KUKA KRL program: EPS_2_25999_MH3A_A_20251114084356.src

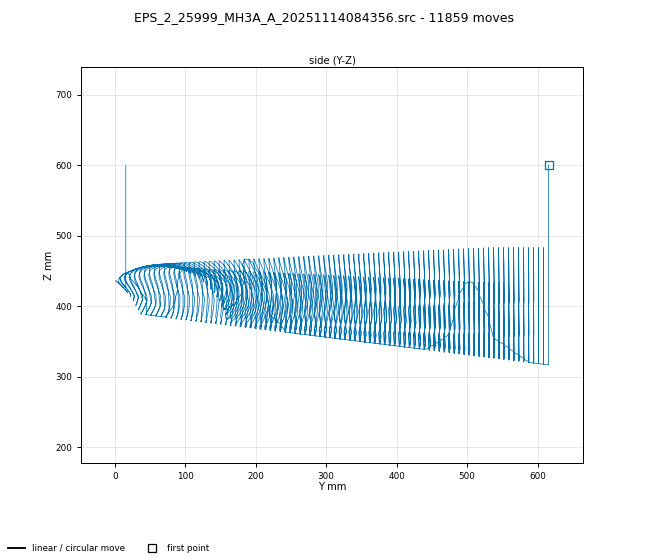
[picture p0: tool path of EPS_2_25999_MH3A_A_20251114084356.src, 11859 of 11861 moves have a stored position in this frame; points joined in program order, loops and branches not executed]
&ACCESS RVP
&REL 4
&COMMENT QRS 19112012
&PARAM EDITMASK = *
DEF PART()
EXT BAS (BAS_COMMAND :IN,REAL :IN )
INT I
BAS (#INITMOV,0 )

;KUKA QRS Post kuka4.cps  Date:22-06-2017 !

File_ID=2914

QRS_PRE_INIT()

;Init var - Until changes are made in qrs_pre_init
Outlet_Square_prg=0
Inlet_1_Square_prg=0
Inlet_2_Square_prg=0
Inlet_3_Square_prg=0
Inlet_4_Square_prg=0
Inlet_5_Square_prg=0

Outlet_1={X 0.000, Y 530.910, Z 408.000, B 0.000, E1 0.000 }
Inlet_1={X 0.000, Y 534.490, Z 358.000, B 0.000, E1 140.000 }
Outlet_1_type=150
Inlet_1_type=150
;QRS#1=Sidecore dimensions
;QRS#2=150-6" PVC SDR 28
;QRS#3=150-6" PVC SDR 28
;QRS#4=
;QRS#5=
;QRS#6=
;QRS#7=
;QRS#8=
;QRS#9=10-06 PSX
;QRS#10=10-06 PSX
;QRS#11=
;QRS#12=
;QRS#13=
;QRS#14=
;QRS#15=
;QRS#16=1220x127x762 2,5'
;QRS#17=EPS Height
;QRS#18=483
;QRS#19=*
;QRS#20= UPDATED VERSION 22-06-2017
;QRS#21=*
Outlet_Square=070
Inlet_1_Square=070
Inlet_2_Square=0
Inlet_3_Square=0
Inlet_4_Square=0
Inlet_5_Square=0
Mill_Square=1
Outlet_Square_Prg=203
Inlet_1_Square_prg=203

QRS_INIT()

$ADVANCE=5

; T1
PTP {E1 173.609,E2 173.609}
PTP {X 0,Y 615.506,A -85,B 0,C 180,E1 173.609,E2 173.609,E3 0,E4 0,E5 0,E6 0}
QRS_SPEED_INIT()
LIN {X 0,Y 615.506,Z 600,A -85,B 0,C 180,E1 173.609,E2 173.609,E3 0,E4 0,E5 0,E6 0} C_VEL
LIN {X 0,Y 615.506,Z 326.684,A -85,B 0,C 180,E1 173.609,E2 173.609} C_VEL
LIN {X 0,Y 615.506,Z 318.507,A -85,B 0,C 180,E1 173.609,E2 173.609} C_VEL
LIN {X 0,Y 615.491,Z 316.507,A -85,B 0,C 180,E1 173.422,E2 173.422} C_VEL
LIN {X 0,Y 615.476,Z 316.513,A -85,B 0,C 180,E1 170.802,E2 170.802} C_VEL
LIN {X 0,Y 615.489,Z 316.515,A -85,B 0,C 180,E1 168.14,E2 168.14} C_VEL
LIN {X 0,Y 615.477,Z 316.512,A -85,B 0,C 180,E1 165.452,E2 165.452} C_VEL
LIN {X 0,Y 615.469,Z 316.512,A -85,B 0,C 180,E1 162.73,E2 162.73} C_VEL
LIN {X 0,Y 615.495,Z 317.045,A -85,B 0,C 180,E1 162.044,E2 162.044} C_VEL
LIN {X 0,Y 615.473,Z 321.165,A -85,B 0,C 180,E1 159.27,E2 159.27} C_VEL
LIN {X 0,Y 615.483,Z 324.407,A -85,B 0,C 180,E1 157.156,E2 157.156} C_VEL
LIN {X 0,Y 615.467,Z 328.675,A -85,B 0,C 180,E1 154.436,E2 154.436} C_VEL
LIN {X 0,Y 615.496,Z 333.308,A -85,B 0,C 180,E1 151.549,E2 151.549} C_VEL
LIN {X 0,Y 615.434,Z 337.615,A -85,B 0,C 180,E1 148.923,E2 148.923} C_VEL
LIN {X 0,Y 615.452,Z 341.695,A -85,B 0,C 180,E1 146.472,E2 146.472} C_VEL
LIN {X 0,Y 615.447,Z 346.56,A -85,B 0,C 180,E1 143.574,E2 143.574} C_VEL
LIN {X 0,Y 615.469,Z 351.05,A -85,B 0,C 180,E1 140.941,E2 140.941} C_VEL
LIN {X 0,Y 615.479,Z 354.222,A -85,B 0,C 180,E1 139.089,E2 139.089} C_VEL
LIN {X 0,Y 615.488,Z 365.834,A -85,B 0,C 180,E1 138.765,E2 138.765} C_VEL
LIN {X 0,Y 615.49,Z 374.096,A -85,B 0,C 180,E1 138.452,E2 138.452} C_VEL
LIN {X 0,Y 615.489,Z 381.984,A -85,B 0,C 180,E1 138.074,E2 138.074} C_VEL
LIN {X 0,Y 615.47,Z 390.539,A -85,B 0,C 180,E1 137.56,E2 137.56} C_VEL
LIN {X 0,Y 615.499,Z 397.606,A -85,B 0,C 180,E1 137.04,E2 137.04} C_VEL
LIN {X 0,Y 615.497,Z 404.982,A -85,B 0,C 180,E1 136.381,E2 136.381} C_VEL
LIN {X 0,Y 615.495,Z 411.606,A -85,B 0,C 180,E1 135.657,E2 135.657} C_VEL
LIN {X 0,Y 615.495,Z 418.335,A -85,B 0,C 180,E1 134.737,E2 134.737} C_VEL
LIN {X 0,Y 615.493,Z 422.558,A -85,B 0,C 180,E1 134,E2 134} C_VEL
LIN {X 0,Y 615.491,Z 426.704,A -85,B 0,C 180,E1 133.049,E2 133.049} C_VEL
LIN {X 0,Y 615.494,Z 429.688,A -85,B 0,C 180,E1 132.082,E2 132.082} C_VEL
LIN {X 0,Y 615.49,Z 431.568,A -85,B 0,C 180,E1 131.097,E2 131.097} C_VEL
LIN {X 0,Y 615.495,Z 432.347,A -85,B 0,C 180,E1 130.092,E2 130.092} C_VEL
LIN {X 0,Y 615.488,Z 431.699,A -85,B 0,C 180,E1 128.905,E2 128.905} C_VEL
LIN {X 0,Y 615.492,Z 430.141,A -85,B 0,C 180,E1 128.014,E2 128.014} C_VEL
LIN {X 0,Y 615.491,Z 426.975,A -85,B 0,C 180,E1 126.939,E2 126.939} C_VEL
LIN {X 0,Y 615.494,Z 422.174,A -85,B 0,C 180,E1 125.837,E2 125.837} C_VEL
LIN {X 0,Y 615.494,Z 417.278,A -85,B 0,C 180,E1 125.015,E2 125.015} C_VEL
LIN {X 0,Y 615.497,Z 411.085,A -85,B 0,C 180,E1 124.192,E2 124.192} C_VEL
LIN {X 0,Y 615.496,Z 405.073,A -85,B 0,C 180,E1 123.538,E2 123.538} C_VEL
LIN {X 0,Y 615.498,Z 398.504,A -85,B 0,C 180,E1 122.943,E2 122.943} C_VEL
LIN {X 0,Y 615.493,Z 392.117,A -85,B 0,C 180,E1 122.458,E2 122.458} C_VEL
LIN {X 0,Y 615.459,Z 385.126,A -85,B 0,C 180,E1 122.01,E2 122.01} C_VEL
LIN {X 0,Y 615.457,Z 375.902,A -85,B 0,C 180,E1 121.538,E2 121.538} C_VEL
LIN {X 0,Y 615.476,Z 367.411,A -85,B 0,C 180,E1 121.199,E2 121.199} C_VEL
LIN {X 0,Y 615.486,Z 359.644,A -85,B 0,C 180,E1 120.962,E2 120.962} C_VEL
LIN {X 0,Y 615.494,Z 354.226,A -85,B 0,C 180,E1 120.825,E2 120.825} C_VEL
LIN {X 0,Y 615.471,Z 349.24,A -85,B 0,C 180,E1 117.917,E2 117.917} C_VEL
LIN {X 0,Y 615.495,Z 345.264,A -85,B 0,C 180,E1 115.573,E2 115.573} C_VEL
LIN {X 0,Y 615.478,Z 340.687,A -85,B 0,C 180,E1 112.846,E2 112.846} C_VEL
LIN {X 0,Y 615.482,Z 336.043,A -85,B 0,C 180,E1 110.034,E2 110.034} C_VEL
LIN {X 0,Y 615.452,Z 332.672,A -85,B 0,C 180,E1 107.959,E2 107.959} C_VEL
LIN {X 0,Y 615.43,Z 329.378,A -85,B 0,C 180,E1 105.907,E2 105.907} C_VEL
LIN {X 0,Y 615.459,Z 325.104,A -85,B 0,C 180,E1 103.203,E2 103.203} C_VEL
LIN {X 0,Y 615.473,Z 320.993,A -85,B 0,C 180,E1 100.528,E2 100.528} C_VEL
LIN {X 0,Y 615.482,Z 317.044,A -85,B 0,C 180,E1 97.876,E2 97.876} C_VEL
LIN {X 0,Y 615.483,Z 316.509,A -85,B 0,C 180,E1 97.216,E2 97.216} C_VEL
LIN {X 0,Y 615.479,Z 316.51,A -85,B 0,C 180,E1 94.585,E2 94.585} C_VEL
LIN {X 0,Y 615.471,Z 316.512,A -85,B 0,C 180,E1 91.964,E2 91.964} C_VEL
LIN {X 0,Y 615.483,Z 316.512,A -85,B 0,C 180,E1 89.347,E2 89.347} C_VEL
LIN {X 0,Y 615.49,Z 316.514,A -85,B 0,C 180,E1 86.728,E2 86.728} C_VEL
LIN {X 0,Y 615.481,Z 316.512,A -85,B 0,C 180,E1 84.102,E2 84.102} C_VEL
LIN {X 0,Y 615.485,Z 316.509,A -85,B 0,C 180,E1 81.464,E2 81.464} C_VEL
LIN {X 0,Y 615.477,Z 316.51,A -85,B 0,C 180,E1 78.808,E2 78.808} C_VEL
LIN {X 0,Y 615.478,Z 316.512,A -85,B 0,C 180,E1 76.066,E2 76.066} C_VEL
LIN {X 0,Y 615.492,Z 316.514,A -85,B 0,C 180,E1 73.415,E2 73.415} C_VEL
LIN {X 0,Y 615.475,Z 316.512,A -85,B 0,C 180,E1 70.663,E2 70.663} C_VEL
LIN {X 0,Y 615.497,Z 316.512,A -85,B 0,C 180,E1 68.57,E2 68.57} C_VEL
LIN {X 0,Y 615.489,Z 316.508,A -85,B 0,C 180,E1 65.729,E2 65.729} C_VEL
LIN {X 0,Y 615.479,Z 316.511,A -85,B 0,C 180,E1 62.824,E2 62.824} C_VEL
LIN {X 0,Y 615.484,Z 316.512,A -85,B 0,C 180,E1 60.204,E2 60.204} C_VEL
LIN {X 0,Y 615.495,Z 316.512,A -85,B 0,C 180,E1 57.544,E2 57.544} C_VEL
LIN {X 0,Y 615.498,Z 316.513,A -85,B 0,C 180,E1 55.187,E2 55.187} C_VEL
LIN {X 0,Y 615.49,Z 316.515,A -85,B 0,C 180,E1 52.759,E2 52.759} C_VEL
LIN {X 0,Y 615.489,Z 316.508,A -85,B 0,C 180,E1 49.909,E2 49.909} C_VEL
LIN {X 0,Y 615.477,Z 316.512,A -85,B 0,C 180,E1 46.952,E2 46.952} C_VEL
LIN {X 0,Y 615.494,Z 316.509,A -85,B 0,C 180,E1 44,E2 44} C_VEL
LIN {X 0,Y 615.468,Z 316.512,A -85,B 0,C 180,E1 41.094,E2 41.094} C_VEL
LIN {X 0,Y 615.467,Z 316.513,A -85,B 0,C 180,E1 38.905,E2 38.905} C_VEL
LIN {X 0,Y 615.474,Z 316.511,A -85,B 0,C 180,E1 36.424,E2 36.424} C_VEL
LIN {X 0,Y 615.492,Z 316.51,A -85,B 0,C 180,E1 33.537,E2 33.537} C_VEL
LIN {X 0,Y 615.491,Z 316.514,A -85,B 0,C 180,E1 30.918,E2 30.918} C_VEL
LIN {X 0,Y 615.496,Z 316.513,A -85,B 0,C 180,E1 28.454,E2 28.454} C_VEL
LIN {X 0,Y 615.466,Z 316.513,A -85,B 0,C 180,E1 25.568,E2 25.568} C_VEL
LIN {X 0,Y 615.468,Z 316.512,A -85,B 0,C 180,E1 22.844,E2 22.844} C_VEL
LIN {X 0,Y 615.493,Z 316.513,A -85,B 0,C 180,E1 20.032,E2 20.032} C_VEL
LIN {X 0,Y 615.476,Z 316.512,A -85,B 0,C 180,E1 17.27,E2 17.27} C_VEL
LIN {X 0,Y 615.485,Z 316.508,A -85,B 0,C 180,E1 14.548,E2 14.548} C_VEL
LIN {X 0,Y 615.484,Z 316.509,A -85,B 0,C 180,E1 11.86,E2 11.86} C_VEL
LIN {X 0,Y 615.483,Z 316.513,A -85,B 0,C 180,E1 9.198,E2 9.198} C_VEL
LIN {X 0,Y 615.494,Z 316.512,A -85,B 0,C 180,E1 6.556,E2 6.556} C_VEL
LIN {X 0,Y 615.477,Z 316.512,A -85,B 0,C 180,E1 3.928,E2 3.928} C_VEL
LIN {X 0,Y 615.468,Z 316.512,A -85,B 0,C 180,E1 1.308,E2 1.308} C_VEL
LIN {X 0,Y 615.49,Z 316.507,A -85,B 0,C 180,E1 -1.309,E2 -1.309} C_VEL
LIN {X 0,Y 615.483,Z 316.51,A -85,B 0,C 180,E1 -3.929,E2 -3.929} C_VEL
LIN {X 0,Y 615.482,Z 316.513,A -85,B 0,C 180,E1 -6.585,E2 -6.585} C_VEL
LIN {X 0,Y 615.496,Z 316.513,A -85,B 0,C 180,E1 -9.199,E2 -9.199} C_VEL
LIN {X 0,Y 615.477,Z 316.512,A -85,B 0,C 180,E1 -11.862,E2 -11.862} C_VEL
LIN {X 0,Y 615.466,Z 316.512,A -85,B 0,C 180,E1 -14.55,E2 -14.55} C_VEL
LIN {X 0,Y 615.496,Z 316.507,A -85,B 0,C 180,E1 -17.271,E2 -17.271} C_VEL
LIN {X 0,Y 615.49,Z 316.513,A -85,B 0,C 180,E1 -20.033,E2 -20.033} C_VEL
LIN {X 0,Y 615.492,Z 316.508,A -85,B 0,C 180,E1 -22.845,E2 -22.845} C_VEL
LIN {X 0,Y 615.472,Z 316.512,A -85,B 0,C 180,E1 -25.717,E2 -25.717} C_VEL
LIN {X 0,Y 615.484,Z 316.513,A -85,B 0,C 180,E1 -28.452,E2 -28.452} C_VEL
LIN {X 0,Y 615.482,Z 316.515,A -85,B 0,C 180,E1 -31.088,E2 -31.088} C_VEL
LIN {X 0,Y 615.491,Z 316.512,A -85,B 0,C 180,E1 -33.537,E2 -33.537} C_VEL
LIN {X 0,Y 615.491,Z 316.514,A -85,B 0,C 180,E1 -35.836,E2 -35.836} C_VEL
LIN {X 0,Y 615.479,Z 316.512,A -85,B 0,C 180,E1 -38.069,E2 -38.069} C_VEL
LIN {X 0,Y 615.48,Z 316.514,A -85,B 0,C 180,E1 -40.607,E2 -40.607} C_VEL
LIN {X 0,Y 615.492,Z 316.512,A -85,B 0,C 180,E1 -43.245,E2 -43.245} C_VEL
LIN {X 0,Y 615.471,Z 316.512,A -85,B 0,C 180,E1 -46.004,E2 -46.004} C_VEL
LIN {X 0,Y 615.493,Z 316.508,A -85,B 0,C 180,E1 -48.905,E2 -48.905} C_VEL
LIN {X 0,Y 615.477,Z 316.51,A -85,B 0,C 180,E1 -51.096,E2 -51.096} C_VEL
LIN {X 0,Y 615.464,Z 316.513,A -85,B 0,C 180,E1 -53.575,E2 -53.575} C_VEL
LIN {X 0,Y 615.466,Z 316.512,A -85,B 0,C 180,E1 -55.978,E2 -55.978} C_VEL
LIN {X 0,Y 615.476,Z 316.691,A -85,B 0,C 180,E1 -57.446,E2 -57.446} C_VEL
LIN {X 0,Y 615.479,Z 325.866,A -85,B 0,C 180,E1 -60.207,E2 -60.207} C_VEL
LIN {X 0,Y 615.441,Z 335.316,A -85,B 0,C 180,E1 -62.964,E2 -62.964} C_VEL
LIN {X 0,Y 615.436,Z 343.744,A -85,B 0,C 180,E1 -65.368,E2 -65.368} C_VEL
LIN {X 0,Y 615.487,Z 352.642,A -85,B 0,C 180,E1 -67.865,E2 -67.865} C_VEL
LIN {X 0,Y 615.467,Z 362.822,A -85,B 0,C 180,E1 -70.662,E2 -70.662} C_VEL
LIN {X 0,Y 615.481,Z 372.986,A -85,B 0,C 180,E1 -73.414,E2 -73.414} C_VEL
LIN {X 0,Y 615.493,Z 383.148,A -85,B 0,C 180,E1 -76.127,E2 -76.127} C_VEL
LIN {X 0,Y 615.48,Z 393.305,A -85,B 0,C 180,E1 -78.808,E2 -78.808} C_VEL
LIN {X 0,Y 615.482,Z 400.916,A -85,B 0,C 180,E1 -80.802,E2 -80.802} C_VEL
LIN {X 0,Y 615.49,Z 414.188,A -85,B 0,C 180,E1 -81.133,E2 -81.133} C_VEL
LIN {X 0,Y 615.472,Z 423.247,A -85,B 0,C 180,E1 -81.464,E2 -81.464} C_VEL
LIN {X 0,Y 615.48,Z 431.93,A -85,B 0,C 180,E1 -81.877,E2 -81.877} C_VEL
LIN {X 0,Y 615.488,Z 440.212,A -85,B 0,C 180,E1 -82.373,E2 -82.373} C_VEL
LIN {X 0,Y 615.499,Z 447.943,A -85,B 0,C 180,E1 -82.943,E2 -82.943} C_VEL
LIN {X 0,Y 615.498,Z 453.655,A -85,B 0,C 180,E1 -83.444,E2 -83.444} C_VEL
LIN {X 0,Y 615.499,Z 459.929,A -85,B 0,C 180,E1 -84.102,E2 -84.102} C_VEL
LIN {X 0,Y 615.495,Z 465.142,A -85,B 0,C 180,E1 -84.76,E2 -84.76} C_VEL
LIN {X 0,Y 615.495,Z 469.487,A -85,B 0,C 180,E1 -85.416,E2 -85.416} C_VEL
LIN {X 0,Y 615.491,Z 474.607,A -85,B 0,C 180,E1 -86.4,E2 -86.4} C_VEL
LIN {X 0,Y 615.488,Z 477.224,A -85,B 0,C 180,E1 -87.056,E2 -87.056} C_VEL
LIN {X 0,Y 615.5,Z 480.087,A -85,B 0,C 180,E1 -88.038,E2 -88.038} C_VEL
LIN {X 0,Y 615.493,Z 481.331,A -85,B 0,C 180,E1 -88.692,E2 -88.692} C_VEL
LIN {X 0,Y 615.491,Z 482.105,A -85,B 0,C 180,E1 -89.347,E2 -89.347} C_VEL
LIN {X 0,Y 615.491,Z 482.389,A -85,B 0,C 180,E1 -90.001,E2 -90.001} C_VEL
LIN {X 0,Y 615.491,Z 482.104,A -85,B 0,C 180,E1 -90.655,E2 -90.655} C_VEL
LIN {X 0,Y 615.493,Z 481.329,A -85,B 0,C 180,E1 -91.309,E2 -91.309} C_VEL
LIN {X 0,Y 615.5,Z 480.083,A -85,B 0,C 180,E1 -91.964,E2 -91.964} C_VEL
LIN {X 0,Y 615.488,Z 477.218,A -85,B 0,C 180,E1 -92.946,E2 -92.946} C_VEL
LIN {X 0,Y 615.491,Z 474.6,A -85,B 0,C 180,E1 -93.601,E2 -93.601} C_VEL
LIN {X 0,Y 615.495,Z 469.478,A -85,B 0,C 180,E1 -94.585,E2 -94.585} C_VEL
LIN {X 0,Y 615.495,Z 463.962,A -85,B 0,C 180,E1 -95.406,E2 -95.406} C_VEL
LIN {X 0,Y 615.498,Z 457.01,A -85,B 0,C 180,E1 -96.228,E2 -96.228} C_VEL
LIN {X 0,Y 615.498,Z 449.854,A -85,B 0,C 180,E1 -96.901,E2 -96.901} C_VEL
LIN {X 0,Y 615.486,Z 442.61,A -85,B 0,C 180,E1 -97.464,E2 -97.464} C_VEL
LIN {X 0,Y 615.487,Z 434.857,A -85,B 0,C 180,E1 -97.959,E2 -97.959} C_VEL
LIN {X 0,Y 615.472,Z 426.902,A -85,B 0,C 180,E1 -98.372,E2 -98.372} C_VEL
LIN {X 0,Y 615.481,Z 417.737,A -85,B 0,C 180,E1 -98.744,E2 -98.744} C_VEL
LIN {X 0,Y 615.492,Z 409.662,A -85,B 0,C 180,E1 -98.992,E2 -98.992} C_VEL
LIN {X 0,Y 615.486,Z 400.908,A -85,B 0,C 180,E1 -99.2,E2 -99.2} C_VEL
LIN {X 0,Y 615.487,Z 390.763,A -85,B 0,C 180,E1 -101.862,E2 -101.862} C_VEL
LIN {X 0,Y 615.489,Z 380.599,A -85,B 0,C 180,E1 -104.55,E2 -104.55} C_VEL
LIN {X 0,Y 615.467,Z 370.447,A -85,B 0,C 180,E1 -107.272,E2 -107.272} C_VEL
LIN {X 0,Y 615.495,Z 360.265,A -85,B 0,C 180,E1 -110.033,E2 -110.033} C_VEL
LIN {X 0,Y 615.465,Z 351.91,A -85,B 0,C 180,E1 -112.341,E2 -112.341} C_VEL
LIN {X 0,Y 615.441,Z 342.46,A -85,B 0,C 180,E1 -114.994,E2 -114.994} C_VEL
LIN {X 0,Y 615.495,Z 333.539,A -85,B 0,C 180,E1 -117.546,E2 -117.546} C_VEL
LIN {X 0,Y 615.496,Z 323.35,A -85,B 0,C 180,E1 -120.539,E2 -120.539} C_VEL
LIN {X 0,Y 615.472,Z 316.513,A -85,B 0,C 180,E1 -122.653,E2 -122.653} C_VEL
LIN {X 0,Y 615.493,Z 316.51,A -85,B 0,C 180,E1 -125.616,E2 -125.616} C_VEL
LIN {X 0,Y 615.494,Z 316.512,A -85,B 0,C 180,E1 -128.069,E2 -128.069} C_VEL
LIN {X 0,Y 615.488,Z 316.508,A -85,B 0,C 180,E1 -131.094,E2 -131.094} C_VEL
LIN {X 0,Y 615.489,Z 316.513,A -85,B 0,C 180,E1 -133.997,E2 -133.997} C_VEL
LIN {X 0,Y 615.487,Z 316.508,A -85,B 0,C 180,E1 -136.953,E2 -136.953} C_VEL
LIN {X 0,Y 615.497,Z 316.512,A -85,B 0,C 180,E1 -139.911,E2 -139.911} C_VEL
LIN {X 0,Y 615.486,Z 316.509,A -85,B 0,C 180,E1 -142.757,E2 -142.757} C_VEL
LIN {X 0,Y 615.489,Z 316.508,A -85,B 0,C 180,E1 -145.3,E2 -145.3} C_VEL
LIN {X 0,Y 615.468,Z 316.513,A -85,B 0,C 180,E1 -147.673,E2 -147.673} C_VEL
LIN {X 0,Y 615.472,Z 316.512,A -85,B 0,C 180,E1 -150.209,E2 -150.209} C_VEL
LIN {X 0,Y 615.498,Z 316.513,A -85,B 0,C 180,E1 -152.954,E2 -152.954} C_VEL
LIN {X 0,Y 615.469,Z 316.513,A -85,B 0,C 180,E1 -155.727,E2 -155.727} C_VEL
LIN {X 0,Y 615.479,Z 316.513,A -85,B 0,C 180,E1 -157.863,E2 -157.863} C_VEL
LIN {X 0,Y 615.491,Z 316.507,A -85,B 0,C 180,E1 -160.662,E2 -160.662} C_VEL
LIN {X 0,Y 615.488,Z 316.515,A -85,B 0,C 180,E1 -163.57,E2 -163.57} C_VEL
LIN {X 0,Y 615.487,Z 316.511,A -85,B 0,C 180,E1 -166.125,E2 -166.125} C_VEL
LIN {X 0,Y 615.485,Z 316.51,A -85,B 0,C 180,E1 -169.115,E2 -169.115} C_VEL
LIN {X 0,Y 615.475,Z 316.512,A -85,B 0,C 180,E1 -171.463,E2 -171.463} C_VEL
LIN {X 0,Y 615.494,Z 316.512,A -85,B 0,C 180,E1 -174.101,E2 -174.101} C_VEL
LIN {X 0,Y 615.484,Z 316.512,A -85,B 0,C 180,E1 -176.726,E2 -176.726} C_VEL
LIN {X 0,Y 615.469,Z 316.512,A -85,B 0,C 180,E1 -179.345,E2 -179.345} C_VEL
LIN {X 0,Y 615.469,Z 316.512,A -85,B 0,C 180,E1 -181.962,E2 -181.962} C_VEL
LIN {X 0,Y 615.497,Z 316.509,A -85,B 0,C 180,E1 -184.584,E2 -184.584} C_VEL
LIN {X 0,Y 615.491,Z 316.507,A -85,B 0,C 180,E1 -186.578,E2 -186.578} C_VEL
LIN {X 0,Y 614.81,Z 316.658,A -85,B 0,C 180,E1 -187.123,E2 -187.123} C_VEL
LIN {X 0,Y 611.969,Z 317.07,A -85,B 0,C 180,E1 -188.009,E2 -188.009} C_VEL
LIN {X 0,Y 609.574,Z 317.381,A -85,B 0,C 180,E1 -188.721,E2 -188.721} C_VEL
LIN {X 0,Y 608.541,Z 317.499,A -85,B 0,C 180,E1 -189.271,E2 -189.271} C_VEL
LIN {X 0,Y 608.453,Z 317.507,A -85,B 0,C 180,E1 -189.457,E2 -189.457} C_VEL
LIN {X 0,Y 608.465,Z 317.508,A -85,B 0,C 180,E1 -191.999,E2 -191.999} C_VEL
LIN {X 0,Y 608.469,Z 317.505,A -85,B 0,C 180,E1 -194.72,E2 -194.72} C_VEL
LIN {X 0,Y 608.445,Z 317.509,A -85,B 0,C 180,E1 -197.476,E2 -197.476} C_VEL
LIN {X 0,Y 608.431,Z 319.28,A -85,B 0,C 180,E1 -198.869,E2 -198.869} C_VEL
LIN {X 0,Y 608.447,Z 323.442,A -85,B 0,C 180,E1 -201.691,E2 -201.691} C_VEL
LIN {X 0,Y 608.425,Z 327.902,A -85,B 0,C 180,E1 -204.571,E2 -204.571} C_VEL
LIN {X 0,Y 608.407,Z 332.056,A -85,B 0,C 180,E1 -207.193,E2 -207.193} C_VEL
LIN {X 0,Y 608.447,Z 336.535,A -85,B 0,C 180,E1 -209.967,E2 -209.967} C_VEL
LIN {X 0,Y 608.385,Z 341.335,A -85,B 0,C 180,E1 -212.883,E2 -212.883} C_VEL
LIN {X 0,Y 608.395,Z 345.335,A -85,B 0,C 180,E1 -215.28,E2 -215.28} C_VEL
LIN {X 0,Y 608.394,Z 350.321,A -85,B 0,C 180,E1 -218.231,E2 -218.231} C_VEL
LIN {X 0,Y 608.429,Z 354.717,A -85,B 0,C 180,E1 -220.807,E2 -220.807} C_VEL
LIN {X 0,Y 608.499,Z 365.683,A -85,B 0,C 180,E1 -221.117,E2 -221.117} C_VEL
LIN {X 0,Y 608.481,Z 375.012,A -85,B 0,C 180,E1 -221.476,E2 -221.476} C_VEL
LIN {X 0,Y 608.478,Z 382.878,A -85,B 0,C 180,E1 -221.864,E2 -221.864} C_VEL
LIN {X 0,Y 608.437,Z 390.587,A -85,B 0,C 180,E1 -222.331,E2 -222.331} C_VEL
LIN {X 0,Y 608.457,Z 397.911,A -85,B 0,C 180,E1 -222.872,E2 -222.872} C_VEL
LIN {X 0,Y 608.475,Z 405.535,A -85,B 0,C 180,E1 -223.558,E2 -223.558} C_VEL
LIN {X 0,Y 608.439,Z 411.929,A -85,B 0,C 180,E1 -224.262,E2 -224.262} C_VEL
LIN {X 0,Y 608.449,Z 418.797,A -85,B 0,C 180,E1 -225.203,E2 -225.203} C_VEL
LIN {X 0,Y 608.43,Z 423.884,A -85,B 0,C 180,E1 -226.126,E2 -226.126} C_VEL
LIN {X 0,Y 608.432,Z 427.69,A -85,B 0,C 180,E1 -227.038,E2 -227.038} C_VEL
LIN {X 0,Y 608.421,Z 430.378,A -85,B 0,C 180,E1 -227.935,E2 -227.935} C_VEL
LIN {X 0,Y 608.426,Z 432.074,A -85,B 0,C 180,E1 -228.82,E2 -228.82} C_VEL
LIN {X 0,Y 608.416,Z 432.859,A -85,B 0,C 180,E1 -229.693,E2 -229.693} C_VEL
LIN {X 0,Y 608.416,Z 432.714,A -85,B 0,C 180,E1 -230.707,E2 -230.707} C_VEL
LIN {X 0,Y 608.421,Z 431.317,A -85,B 0,C 180,E1 -231.763,E2 -231.763} C_VEL
LIN {X 0,Y 608.432,Z 428.408,A -85,B 0,C 180,E1 -232.844,E2 -232.844} C_VEL
LIN {X 0,Y 608.453,Z 426.016,A -85,B 0,C 180,E1 -233.497,E2 -233.497} C_VEL
LIN {X 0,Y 608.445,Z 420.866,A -85,B 0,C 180,E1 -234.53,E2 -234.53} C_VEL
LIN {X 0,Y 608.442,Z 415.856,A -85,B 0,C 180,E1 -235.312,E2 -235.312} C_VEL
LIN {X 0,Y 608.443,Z 409.395,A -85,B 0,C 180,E1 -236.125,E2 -236.125} C_VEL
LIN {X 0,Y 608.453,Z 401.492,A -85,B 0,C 180,E1 -236.922,E2 -236.922} C_VEL
LIN {X 0,Y 608.48,Z 393.219,A -85,B 0,C 180,E1 -237.578,E2 -237.578} C_VEL
LIN {X 0,Y 608.432,Z 385.171,A -85,B 0,C 180,E1 -238.098,E2 -238.098} C_VEL
LIN {X 0,Y 608.44,Z 376.755,A -85,B 0,C 180,E1 -238.536,E2 -238.536} C_VEL
LIN {X 0,Y 608.488,Z 367.056,A -85,B 0,C 180,E1 -238.926,E2 -238.926} C_VEL
LIN {X 0,Y 608.503,Z 358.051,A -85,B 0,C 180,E1 -239.192,E2 -239.192} C_VEL
LIN {X 0,Y 608.449,Z 354.713,A -85,B 0,C 180,E1 -239.285,E2 -239.285} C_VEL
LIN {X 0,Y 608.429,Z 350.537,A -85,B 0,C 180,E1 -241.732,E2 -241.732} C_VEL
LIN {X 0,Y 608.43,Z 345.523,A -85,B 0,C 180,E1 -244.697,E2 -244.697} C_VEL
LIN {X 0,Y 608.425,Z 340.695,A -85,B 0,C 180,E1 -247.592,E2 -247.592} C_VEL
LIN {X 0,Y 608.408,Z 336.041,A -85,B 0,C 180,E1 -250.427,E2 -250.427} C_VEL
LIN {X 0,Y 608.436,Z 331.546,A -85,B 0,C 180,E1 -253.215,E2 -253.215} C_VEL
LIN {X 0,Y 608.37,Z 327.129,A -85,B 0,C 180,E1 -256.015,E2 -256.015} C_VEL
LIN {X 0,Y 608.441,Z 323.04,A -85,B 0,C 180,E1 -258.675,E2 -258.675} C_VEL
LIN {X 0,Y 608.449,Z 319.036,A -85,B 0,C 180,E1 -261.363,E2 -261.363} C_VEL
LIN {X 0,Y 608.439,Z 318.049,A -85,B 0,C 180,E1 -262.032,E2 -262.032} C_VEL
LIN {X 0,Y 608.444,Z 317.508,A -85,B 0,C 180,E1 -262.7,E2 -262.7} C_VEL
LIN {X 0,Y 608.448,Z 317.507,A -85,B 0,C 180,E1 -265.361,E2 -265.361} C_VEL
LIN {X 0,Y 608.441,Z 317.509,A -85,B 0,C 180,E1 -268.013,E2 -268.013} C_VEL
LIN {X 0,Y 608.477,Z 317.506,A -85,B 0,C 180,E1 -270.661,E2 -270.661} C_VEL
LIN {X 0,Y 608.48,Z 317.507,A -85,B 0,C 180,E1 -273.31,E2 -273.31} C_VEL
LIN {X 0,Y 608.453,Z 317.508,A -85,B 0,C 180,E1 -275.966,E2 -275.966} C_VEL
LIN {X 0,Y 608.455,Z 317.506,A -85,B 0,C 180,E1 -278.635,E2 -278.635} C_VEL
LIN {X 0,Y 608.467,Z 317.505,A -85,B 0,C 180,E1 -281.323,E2 -281.323} C_VEL
LIN {X 0,Y 608.456,Z 317.509,A -85,B 0,C 180,E1 -284.037,E2 -284.037} C_VEL
LIN {X 0,Y 608.47,Z 317.507,A -85,B 0,C 180,E1 -286.783,E2 -286.783} C_VEL
LIN {X 0,Y 608.442,Z 317.508,A -85,B 0,C 180,E1 -289.57,E2 -289.57} C_VEL
LIN {X 0,Y 608.461,Z 317.507,A -85,B 0,C 180,E1 -292.405,E2 -292.405} C_VEL
LIN {X 0,Y 608.456,Z 317.506,A -85,B 0,C 180,E1 -294.57,E2 -294.57} C_VEL
LIN {X 0,Y 608.441,Z 317.512,A -85,B 0,C 180,E1 -297.517,E2 -297.517} C_VEL
LIN {X 0,Y 608.467,Z 317.509,A -85,B 0,C 180,E1 -299.974,E2 -299.974} C_VEL
LIN {X 0,Y 608.465,Z 317.508,A -85,B 0,C 180,E1 -302.525,E2 -302.525} C_VEL
LIN {X 0,Y 608.437,Z 317.509,A -85,B 0,C 180,E1 -305.277,E2 -305.277} C_VEL
LIN {X 0,Y 608.463,Z 317.506,A -85,B 0,C 180,E1 -307.745,E2 -307.745} C_VEL
LIN {X 0,Y 608.466,Z 317.505,A -85,B 0,C 180,E1 -310.332,E2 -310.332} C_VEL
LIN {X 0,Y 608.446,Z 317.508,A -85,B 0,C 180,E1 -312.959,E2 -312.959} C_VEL
LIN {X 0,Y 608.46,Z 317.51,A -85,B 0,C 180,E1 -315.734,E2 -315.734} C_VEL
LIN {X 0,Y 608.447,Z 317.508,A -85,B 0,C 180,E1 -318.658,E2 -318.658} C_VEL
LIN {X 0,Y 608.459,Z 317.506,A -85,B 0,C 180,E1 -321.413,E2 -321.413} C_VEL
LIN {X 0,Y 608.468,Z 317.506,A -85,B 0,C 180,E1 -323.95,E2 -323.95} C_VEL
LIN {X 0,Y 608.469,Z 317.505,A -85,B 0,C 180,E1 -326.331,E2 -326.331} C_VEL
LIN {X 0,Y 608.465,Z 317.506,A -85,B 0,C 180,E1 -328.727,E2 -328.727} C_VEL
LIN {X 0,Y 608.47,Z 317.507,A -85,B 0,C 180,E1 -331.378,E2 -331.378} C_VEL
LIN {X 0,Y 608.431,Z 317.514,A -85,B 0,C 180,E1 -333.965,E2 -333.965} C_VEL
LIN {X 0,Y 608.471,Z 317.506,A -85,B 0,C 180,E1 -336.156,E2 -336.156} C_VEL
LIN {X 0,Y 608.469,Z 317.505,A -85,B 0,C 180,E1 -338.309,E2 -338.309} C_VEL
LIN {X 0,Y 608.468,Z 317.509,A -85,B 0,C 180,E1 -341.281,E2 -341.281} C_VEL
LIN {X 0,Y 608.453,Z 317.508,A -85,B 0,C 180,E1 -343.907,E2 -343.907} C_VEL
LIN {X 0,Y 608.449,Z 317.507,A -85,B 0,C 180,E1 -346.644,E2 -346.644} C_VEL
LIN {X 0,Y 608.456,Z 317.507,A -85,B 0,C 180,E1 -349.351,E2 -349.351} C_VEL
LIN {X 0,Y 608.478,Z 317.506,A -85,B 0,C 180,E1 -352.034,E2 -352.034} C_VEL
LIN {X 0,Y 608.465,Z 317.508,A -85,B 0,C 180,E1 -354.699,E2 -354.699} C_VEL
LIN {X 0,Y 608.483,Z 317.504,A -85,B 0,C 180,E1 -357.353,E2 -357.353} C_VEL
LIN {X 0,Y 608.461,Z 317.506,A -85,B 0,C 180,E1 -360.001,E2 -360.001} C_VEL
LIN {X 0,Y 608.46,Z 317.506,A -85,B 0,C 180,E1 -362.649,E2 -362.649} C_VEL
LIN {X 0,Y 608.463,Z 317.507,A -85,B 0,C 180,E1 -365.302,E2 -365.302} C_VEL
LIN {X 0,Y 608.475,Z 317.508,A -85,B 0,C 180,E1 -367.968,E2 -367.968} C_VEL
LIN {X 0,Y 608.464,Z 317.507,A -85,B 0,C 180,E1 -370.65,E2 -370.65} C_VEL
LIN {X 0,Y 608.472,Z 317.504,A -85,B 0,C 180,E1 -373.357,E2 -373.357} C_VEL
LIN {X 0,Y 608.449,Z 317.508,A -85,B 0,C 180,E1 -376.095,E2 -376.095} C_VEL
LIN {X 0,Y 608.449,Z 317.511,A -85,B 0,C 180,E1 -378.87,E2 -378.87} C_VEL
LIN {X 0,Y 608.463,Z 317.506,A -85,B 0,C 180,E1 -381.692,E2 -381.692} C_VEL
LIN {X 0,Y 608.446,Z 317.508,A -85,B 0,C 180,E1 -384.572,E2 -384.572} C_VEL
LIN {X 0,Y 608.486,Z 317.505,A -85,B 0,C 180,E1 -387.212,E2 -387.212} C_VEL
LIN {X 0,Y 608.47,Z 317.507,A -85,B 0,C 180,E1 -389.974,E2 -389.974} C_VEL
LIN {X 0,Y 608.462,Z 317.506,A -85,B 0,C 180,E1 -392.88,E2 -392.88} C_VEL
LIN {X 0,Y 608.444,Z 317.508,A -85,B 0,C 180,E1 -395.278,E2 -395.278} C_VEL
LIN {X 0,Y 608.462,Z 317.506,A -85,B 0,C 180,E1 -397.747,E2 -397.747} C_VEL
LIN {X 0,Y 608.437,Z 317.509,A -85,B 0,C 180,E1 -400.329,E2 -400.329} C_VEL
LIN {X 0,Y 608.456,Z 317.508,A -85,B 0,C 180,E1 -402.96,E2 -402.96} C_VEL
LIN {X 0,Y 608.449,Z 317.51,A -85,B 0,C 180,E1 -405.737,E2 -405.737} C_VEL
LIN {X 0,Y 608.466,Z 317.508,A -85,B 0,C 180,E1 -407.941,E2 -407.941} C_VEL
LIN {X 0,Y 608.47,Z 317.506,A -85,B 0,C 180,E1 -410.703,E2 -410.703} C_VEL
LIN {X 0,Y 608.447,Z 317.509,A -85,B 0,C 180,E1 -413.086,E2 -413.086} C_VEL
LIN {X 0,Y 608.467,Z 317.507,A -85,B 0,C 180,E1 -415.532,E2 -415.532} C_VEL
LIN {X 0,Y 608.461,Z 317.545,A -85,B 0,C 180,E1 -417.28,E2 -417.28} C_VEL
LIN {X 0,Y 608.517,Z 324.656,A -85,B 0,C 180,E1 -419.459,E2 -419.459} C_VEL
LIN {X 0,Y 608.475,Z 333.607,A -85,B 0,C 180,E1 -422.111,E2 -422.111} C_VEL
LIN {X 0,Y 608.45,Z 342.549,A -85,B 0,C 180,E1 -424.7,E2 -424.7} C_VEL
LIN {X 0,Y 608.456,Z 352.516,A -85,B 0,C 180,E1 -427.525,E2 -427.525} C_VEL
LIN {X 0,Y 608.454,Z 362.986,A -85,B 0,C 180,E1 -430.431,E2 -430.431} C_VEL
LIN {X 0,Y 608.439,Z 373.205,A -85,B 0,C 180,E1 -433.217,E2 -433.217} C_VEL
LIN {X 0,Y 608.439,Z 383.542,A -85,B 0,C 180,E1 -435.995,E2 -435.995} C_VEL
LIN {X 0,Y 608.447,Z 393.642,A -85,B 0,C 180,E1 -438.677,E2 -438.677} C_VEL
LIN {X 0,Y 608.422,Z 401.306,A -85,B 0,C 180,E1 -440.694,E2 -440.694} C_VEL
LIN {X 0,Y 608.495,Z 414.508,A -85,B 0,C 180,E1 -441.031,E2 -441.031} C_VEL
LIN {X 0,Y 608.472,Z 423.555,A -85,B 0,C 180,E1 -441.365,E2 -441.365} C_VEL
LIN {X 0,Y 608.459,Z 432.249,A -85,B 0,C 180,E1 -441.783,E2 -441.783} C_VEL
LIN {X 0,Y 608.466,Z 440.555,A -85,B 0,C 180,E1 -442.284,E2 -442.284} C_VEL
LIN {X 0,Y 608.464,Z 448.412,A -85,B 0,C 180,E1 -442.868,E2 -442.868} C_VEL
LIN {X 0,Y 608.466,Z 455.363,A -85,B 0,C 180,E1 -443.496,E2 -443.496} C_VEL
LIN {X 0,Y 608.469,Z 463.198,A -85,B 0,C 180,E1 -444.367,E2 -444.367} C_VEL
LIN {X 0,Y 608.448,Z 469.032,A -85,B 0,C 180,E1 -445.197,E2 -445.197} C_VEL
LIN {X 0,Y 608.434,Z 473.635,A -85,B 0,C 180,E1 -446.027,E2 -446.027} C_VEL
LIN {X 0,Y 608.423,Z 476.625,A -85,B 0,C 180,E1 -446.69,E2 -446.69} C_VEL
LIN {X 0,Y 608.423,Z 478.934,A -85,B 0,C 180,E1 -447.353,E2 -447.353} C_VEL
LIN {X 0,Y 608.444,Z 480.68,A -85,B 0,C 180,E1 -448.015,E2 -448.015} C_VEL
LIN {X 0,Y 608.446,Z 481.935,A -85,B 0,C 180,E1 -448.677,E2 -448.677} C_VEL
LIN {X 0,Y 608.434,Z 482.714,A -85,B 0,C 180,E1 -449.339,E2 -449.339} C_VEL
LIN {X 0,Y 608.431,Z 483,A -85,B 0,C 180,E1 -450.001,E2 -450.001} C_VEL
LIN {X 0,Y 608.434,Z 482.713,A -85,B 0,C 180,E1 -450.663,E2 -450.663} C_VEL
LIN {X 0,Y 608.445,Z 481.932,A -85,B 0,C 180,E1 -451.325,E2 -451.325} C_VEL
LIN {X 0,Y 608.444,Z 480.676,A -85,B 0,C 180,E1 -451.987,E2 -451.987} C_VEL
LIN {X 0,Y 608.444,Z 477.783,A -85,B 0,C 180,E1 -452.98,E2 -452.98} C_VEL
LIN {X 0,Y 608.445,Z 475.142,A -85,B 0,C 180,E1 -453.643,E2 -453.643} C_VEL
LIN {X 0,Y 608.431,Z 469.98,A -85,B 0,C 180,E1 -454.639,E2 -454.639} C_VEL
LIN {X 0,Y 608.46,Z 464.424,A -85,B 0,C 180,E1 -455.469,E2 -455.469} C_VEL
LIN {X 0,Y 608.455,Z 456.672,A -85,B 0,C 180,E1 -456.375,E2 -456.375} C_VEL
LIN {X 0,Y 608.456,Z 449.405,A -85,B 0,C 180,E1 -457.05,E2 -457.05} C_VEL
LIN {X 0,Y 608.468,Z 441.748,A -85,B 0,C 180,E1 -457.634,E2 -457.634} C_VEL
LIN {X 0,Y 608.481,Z 433.705,A -85,B 0,C 180,E1 -458.135,E2 -458.135} C_VEL
LIN {X 0,Y 608.479,Z 425.371,A -85,B 0,C 180,E1 -458.553,E2 -458.553} C_VEL
LIN {X 0,Y 608.484,Z 416.865,A -85,B 0,C 180,E1 -458.888,E2 -458.888} C_VEL
LIN {X 0,Y 608.507,Z 407.553,A -85,B 0,C 180,E1 -459.159,E2 -459.159} C_VEL
LIN {X 0,Y 608.425,Z 401.299,A -85,B 0,C 180,E1 -459.307,E2 -459.307} C_VEL
LIN {X 0,Y 608.429,Z 391.081,A -85,B 0,C 180,E1 -462.001,E2 -462.001} C_VEL
LIN {X 0,Y 608.444,Z 380.862,A -85,B 0,C 180,E1 -464.722,E2 -464.722} C_VEL
LIN {X 0,Y 608.455,Z 370.643,A -85,B 0,C 180,E1 -467.477,E2 -467.477} C_VEL
LIN {X 0,Y 608.455,Z 360.425,A -85,B 0,C 180,E1 -470.275,E2 -470.275} C_VEL
LIN {X 0,Y 608.425,Z 351.485,A -85,B 0,C 180,E1 -472.766,E2 -472.766} C_VEL
LIN {X 0,Y 608.45,Z 342.542,A -85,B 0,C 180,E1 -475.302,E2 -475.302} C_VEL
LIN {X 0,Y 608.475,Z 333.601,A -85,B 0,C 180,E1 -477.891,E2 -477.891} C_VEL
LIN {X 0,Y 608.518,Z 324.639,A -85,B 0,C 180,E1 -480.543,E2 -480.543} C_VEL
LIN {X 0,Y 608.452,Z 317.508,A -85,B 0,C 180,E1 -482.775,E2 -482.775} C_VEL
LIN {X 0,Y 608.447,Z 317.508,A -85,B 0,C 180,E1 -485.278,E2 -485.278} C_VEL
LIN {X 0,Y 608.475,Z 317.504,A -85,B 0,C 180,E1 -487.746,E2 -487.746} C_VEL
LIN {X 0,Y 608.445,Z 317.51,A -85,B 0,C 180,E1 -490.328,E2 -490.328} C_VEL
LIN {X 0,Y 608.485,Z 317.503,A -85,B 0,C 180,E1 -493.31,E2 -493.31} C_VEL
LIN {X 0,Y 608.459,Z 317.507,A -85,B 0,C 180,E1 -496.129,E2 -496.129} C_VEL
LIN {X 0,Y 608.457,Z 317.51,A -85,B 0,C 180,E1 -498.823,E2 -498.823} C_VEL
LIN {X 0,Y 608.457,Z 317.506,A -85,B 0,C 180,E1 -501.762,E2 -501.762} C_VEL
LIN {X 0,Y 608.445,Z 317.508,A -85,B 0,C 180,E1 -503.955,E2 -503.955} C_VEL
LIN {X 0,Y 608.448,Z 317.508,A -85,B 0,C 180,E1 -506.328,E2 -506.328} C_VEL
LIN {X 0,Y 608.452,Z 317.507,A -85,B 0,C 180,E1 -508.732,E2 -508.732} C_VEL
LIN {X 0,Y 608.474,Z 317.505,A -85,B 0,C 180,E1 -511.381,E2 -511.381} C_VEL
LIN {X 0,Y 608.439,Z 317.511,A -85,B 0,C 180,E1 -513.964,E2 -513.964} C_VEL
LIN {X 0,Y 608.456,Z 317.507,A -85,B 0,C 180,E1 -516.154,E2 -516.154} C_VEL
LIN {X 0,Y 608.46,Z 317.506,A -85,B 0,C 180,E1 -518.308,E2 -518.308} C_VEL
LIN {X 0,Y 608.471,Z 317.508,A -85,B 0,C 180,E1 -521.285,E2 -521.285} C_VEL
LIN {X 0,Y 608.451,Z 317.508,A -85,B 0,C 180,E1 -523.905,E2 -523.905} C_VEL
LIN {X 0,Y 608.473,Z 317.505,A -85,B 0,C 180,E1 -526.643,E2 -526.643} C_VEL
LIN {X 0,Y 608.466,Z 317.508,A -85,B 0,C 180,E1 -529.35,E2 -529.35} C_VEL
LIN {X 0,Y 608.477,Z 317.505,A -85,B 0,C 180,E1 -532.032,E2 -532.032} C_VEL
LIN {X 0,Y 608.471,Z 317.505,A -85,B 0,C 180,E1 -534.698,E2 -534.698} C_VEL
LIN {X 0,Y 608.465,Z 317.506,A -85,B 0,C 180,E1 -537.351,E2 -537.351} C_VEL
LIN {X 0,Y 608.478,Z 317.507,A -85,B 0,C 180,E1 -539.999,E2 -539.999} C_VEL
LIN {X 0,Y 608.477,Z 317.505,A -85,B 0,C 180,E1 -542.647,E2 -542.647} C_VEL
LIN {X 0,Y 608.452,Z 317.507,A -85,B 0,C 180,E1 -545.301,E2 -545.301} C_VEL
LIN {X 0,Y 608.464,Z 317.508,A -85,B 0,C 180,E1 -547.299,E2 -547.299} C_VEL
LIN {X 0,Y 608.453,Z 317.507,A -85,B 0,C 180,E1 -549.457,E2 -549.457} C_VEL
LIN {X 0,Y 607.779,Z 317.591,A -85,B 0,C 180,E1 -550.01,E2 -550.01} C_VEL
LIN {X 0,Y 604.929,Z 317.947,A -85,B 0,C 180,E1 -550.907,E2 -550.907} C_VEL
LIN {X 0,Y 602.527,Z 318.247,A -85,B 0,C 180,E1 -551.628,E2 -551.628} C_VEL
LIN {X 0,Y 601.496,Z 318.375,A -85,B 0,C 180,E1 -552.185,E2 -552.185} C_VEL
LIN {X 0,Y 601.412,Z 318.384,A -85,B 0,C 180,E1 -552.373,E2 -552.373} C_VEL
LIN {X 0,Y 601.426,Z 318.383,A -85,B 0,C 180,E1 -554.896,E2 -554.896} C_VEL
LIN {X 0,Y 601.422,Z 318.383,A -85,B 0,C 180,E1 -556.985,E2 -556.985} C_VEL
LIN {X 0,Y 601.392,Z 318.39,A -85,B 0,C 180,E1 -557.688,E2 -557.688} C_VEL
LIN {X 0,Y 601.381,Z 321.316,A -85,B 0,C 180,E1 -559.809,E2 -559.809} C_VEL
LIN {X 0,Y 601.365,Z 325.51,A -85,B 0,C 180,E1 -562.684,E2 -562.684} C_VEL
LIN {X 0,Y 601.343,Z 328.879,A -85,B 0,C 180,E1 -564.88,E2 -564.88} C_VEL
LIN {X 0,Y 601.329,Z 332.746,A -85,B 0,C 180,E1 -567.346,E2 -567.346} C_VEL
LIN {X 0,Y 601.345,Z 337.257,A -85,B 0,C 180,E1 -570.167,E2 -570.167} C_VEL
LIN {X 0,Y 601.316,Z 341.375,A -85,B 0,C 180,E1 -572.699,E2 -572.699} C_VEL
LIN {X 0,Y 601.284,Z 345.327,A -85,B 0,C 180,E1 -575.096,E2 -575.096} C_VEL
LIN {X 0,Y 601.314,Z 349.209,A -85,B 0,C 180,E1 -577.427,E2 -577.427} C_VEL
LIN {X 0,Y 601.299,Z 353.543,A -85,B 0,C 180,E1 -580.003,E2 -580.003} C_VEL
LIN {X 0,Y 601.331,Z 354.732,A -85,B 0,C 180,E1 -580.704,E2 -580.704} C_VEL
LIN {X 0,Y 601.493,Z 364.704,A -85,B 0,C 180,E1 -580.977,E2 -580.977} C_VEL
LIN {X 0,Y 601.483,Z 373.612,A -85,B 0,C 180,E1 -581.311,E2 -581.311} C_VEL
LIN {X 0,Y 601.446,Z 382.782,A -85,B 0,C 180,E1 -581.762,E2 -581.762} C_VEL
LIN {X 0,Y 601.389,Z 391.616,A -85,B 0,C 180,E1 -582.311,E2 -582.311} C_VEL
LIN {X 0,Y 601.422,Z 399.213,A -85,B 0,C 180,E1 -582.896,E2 -582.896} C_VEL
LIN {X 0,Y 601.412,Z 407.729,A -85,B 0,C 180,E1 -583.702,E2 -583.702} C_VEL
LIN {X 0,Y 601.393,Z 414.562,A -85,B 0,C 180,E1 -584.531,E2 -584.531} C_VEL
LIN {X 0,Y 601.374,Z 419.188,A -85,B 0,C 180,E1 -585.213,E2 -585.213} C_VEL
LIN {X 0,Y 601.349,Z 424.31,A -85,B 0,C 180,E1 -586.174,E2 -586.174} C_VEL
LIN {X 0,Y 601.333,Z 427.272,A -85,B 0,C 180,E1 -586.88,E2 -586.88} C_VEL
LIN {X 0,Y 601.356,Z 430.171,A -85,B 0,C 180,E1 -587.823,E2 -587.823} C_VEL
LIN {X 0,Y 601.319,Z 431.522,A -85,B 0,C 180,E1 -588.416,E2 -588.416} C_VEL
LIN {X 0,Y 601.315,Z 432.742,A -85,B 0,C 180,E1 -589.436,E2 -589.436} C_VEL
LIN {X 0,Y 601.301,Z 432.995,A -85,B 0,C 180,E1 -589.995,E2 -589.995} C_VEL
LIN {X 0,Y 601.309,Z 432.627,A -85,B 0,C 180,E1 -590.865,E2 -590.865} C_VEL
LIN {X 0,Y 601.332,Z 431.434,A -85,B 0,C 180,E1 -591.725,E2 -591.725} C_VEL
LIN {X 0,Y 601.328,Z 429.249,A -85,B 0,C 180,E1 -592.629,E2 -592.629} C_VEL
LIN {X 0,Y 601.354,Z 426.551,A -85,B 0,C 180,E1 -593.413,E2 -593.413} C_VEL
LIN {X 0,Y 601.351,Z 422.791,A -85,B 0,C 180,E1 -594.242,E2 -594.242} C_VEL
LIN {X 0,Y 601.37,Z 418.022,A -85,B 0,C 180,E1 -595.064,E2 -595.064} C_VEL
LIN {X 0,Y 601.391,Z 412.08,A -85,B 0,C 180,E1 -595.879,E2 -595.879} C_VEL
LIN {X 0,Y 601.401,Z 404.77,A -85,B 0,C 180,E1 -596.684,E2 -596.684} C_VEL
LIN {X 0,Y 601.422,Z 397.481,A -85,B 0,C 180,E1 -597.338,E2 -597.338} C_VEL
LIN {X 0,Y 601.399,Z 388.753,A -85,B 0,C 180,E1 -597.977,E2 -597.977} C_VEL
LIN {X 0,Y 601.423,Z 378.799,A -85,B 0,C 180,E1 -598.543,E2 -598.543} C_VEL
LIN {X 0,Y 601.468,Z 368.585,A -85,B 0,C 180,E1 -598.977,E2 -598.977} C_VEL
LIN {X 0,Y 601.474,Z 359.309,A -85,B 0,C 180,E1 -599.268,E2 -599.268} C_VEL
LIN {X 0,Y 601.335,Z 354.716,A -85,B 0,C 180,E1 -599.393,E2 -599.393} C_VEL
LIN {X 0,Y 601.323,Z 350.108,A -85,B 0,C 180,E1 -602.127,E2 -602.127} C_VEL
LIN {X 0,Y 601.337,Z 345.119,A -85,B 0,C 180,E1 -605.118,E2 -605.118} C_VEL
LIN {X 0,Y 601.348,Z 341.347,A -85,B 0,C 180,E1 -607.407,E2 -607.407} C_VEL
LIN {X 0,Y 601.316,Z 336.832,A -85,B 0,C 180,E1 -610.187,E2 -610.187} C_VEL
LIN {X 0,Y 601.339,Z 332.324,A -85,B 0,C 180,E1 -613.011,E2 -613.011} C_VEL
LIN {X 0,Y 601.303,Z 327.738,A -85,B 0,C 180,E1 -615.948,E2 -615.948} C_VEL
LIN {X 0,Y 601.389,Z 323.175,A -85,B 0,C 180,E1 -618.999,E2 -618.999} C_VEL
LIN {X 0,Y 601.382,Z 318.828,A -85,B 0,C 180,E1 -621.938,E2 -621.938} C_VEL
LIN {X 0,Y 601.387,Z 318.388,A -85,B 0,C 180,E1 -622.613,E2 -622.613} C_VEL
LIN {X 0,Y 601.418,Z 318.383,A -85,B 0,C 180,E1 -625.307,E2 -625.307} C_VEL
LIN {X 0,Y 601.412,Z 318.384,A -85,B 0,C 180,E1 -627.99,E2 -627.99} C_VEL
LIN {X 0,Y 601.447,Z 318.382,A -85,B 0,C 180,E1 -630.669,E2 -630.669} C_VEL
LIN {X 0,Y 601.43,Z 318.384,A -85,B 0,C 180,E1 -633.349,E2 -633.349} C_VEL
LIN {X 0,Y 601.406,Z 318.385,A -85,B 0,C 180,E1 -636.036,E2 -636.036} C_VEL
LIN {X 0,Y 601.435,Z 318.381,A -85,B 0,C 180,E1 -638.737,E2 -638.737} C_VEL
LIN {X 0,Y 601.426,Z 318.383,A -85,B 0,C 180,E1 -641.457,E2 -641.457} C_VEL
LIN {X 0,Y 601.409,Z 318.388,A -85,B 0,C 180,E1 -644.205,E2 -644.205} C_VEL
LIN {X 0,Y 601.424,Z 318.383,A -85,B 0,C 180,E1 -646.985,E2 -646.985} C_VEL
LIN {X 0,Y 601.399,Z 318.386,A -85,B 0,C 180,E1 -649.809,E2 -649.809} C_VEL
LIN {X 0,Y 601.402,Z 318.388,A -85,B 0,C 180,E1 -652.605,E2 -652.605} C_VEL
LIN {X 0,Y 601.4,Z 318.387,A -85,B 0,C 180,E1 -654.877,E2 -654.877} C_VEL
LIN {X 0,Y 601.416,Z 318.384,A -85,B 0,C 180,E1 -657.866,E2 -657.866} C_VEL
LIN {X 0,Y 601.435,Z 318.383,A -85,B 0,C 180,E1 -660.162,E2 -660.162} C_VEL
LIN {X 0,Y 601.421,Z 318.384,A -85,B 0,C 180,E1 -662.717,E2 -662.717} C_VEL
LIN {X 0,Y 601.409,Z 318.385,A -85,B 0,C 180,E1 -665.116,E2 -665.116} C_VEL
LIN {X 0,Y 601.424,Z 318.384,A -85,B 0,C 180,E1 -667.418,E2 -667.418} C_VEL
LIN {X 0,Y 601.409,Z 318.385,A -85,B 0,C 180,E1 -669.994,E2 -669.994} C_VEL
LIN {X 0,Y 601.426,Z 318.382,A -85,B 0,C 180,E1 -672.667,E2 -672.667} C_VEL
LIN {X 0,Y 601.41,Z 318.385,A -85,B 0,C 180,E1 -675.482,E2 -675.482} C_VEL
LIN {X 0,Y 601.411,Z 318.386,A -85,B 0,C 180,E1 -678.406,E2 -678.406} C_VEL
LIN {X 0,Y 601.425,Z 318.383,A -85,B 0,C 180,E1 -680.876,E2 -680.876} C_VEL
LIN {X 0,Y 601.434,Z 318.381,A -85,B 0,C 180,E1 -683.733,E2 -683.733} C_VEL
LIN {X 0,Y 601.425,Z 318.386,A -85,B 0,C 180,E1 -686.688,E2 -686.688} C_VEL
LIN {X 0,Y 601.424,Z 318.386,A -85,B 0,C 180,E1 -689.059,E2 -689.059} C_VEL
LIN {X 0,Y 601.429,Z 318.384,A -85,B 0,C 180,E1 -691.374,E2 -691.374} C_VEL
LIN {X 0,Y 601.39,Z 318.387,A -85,B 0,C 180,E1 -693.637,E2 -693.637} C_VEL
LIN {X 0,Y 601.46,Z 318.378,A -85,B 0,C 180,E1 -695.861,E2 -695.861} C_VEL
LIN {X 0,Y 601.411,Z 318.384,A -85,B 0,C 180,E1 -698.042,E2 -698.042} C_VEL
LIN {X 0,Y 601.398,Z 318.388,A -85,B 0,C 180,E1 -700.191,E2 -700.191} C_VEL
LIN {X 0,Y 601.422,Z 318.383,A -85,B 0,C 180,E1 -703.015,E2 -703.015} C_VEL
LIN {X 0,Y 601.412,Z 318.386,A -85,B 0,C 180,E1 -705.907,E2 -705.907} C_VEL
LIN {X 0,Y 601.426,Z 318.386,A -85,B 0,C 180,E1 -708.543,E2 -708.543} C_VEL
LIN {X 0,Y 601.434,Z 318.382,A -85,B 0,C 180,E1 -711.263,E2 -711.263} C_VEL
LIN {X 0,Y 601.405,Z 318.385,A -85,B 0,C 180,E1 -713.964,E2 -713.964} C_VEL
LIN {X 0,Y 601.419,Z 318.383,A -85,B 0,C 180,E1 -716.651,E2 -716.651} C_VEL
LIN {X 0,Y 601.447,Z 318.382,A -85,B 0,C 180,E1 -719.331,E2 -719.331} C_VEL
LIN {X 0,Y 601.428,Z 318.384,A -85,B 0,C 180,E1 -722.01,E2 -722.01} C_VEL
LIN {X 0,Y 601.416,Z 318.384,A -85,B 0,C 180,E1 -724.693,E2 -724.693} C_VEL
LIN {X 0,Y 601.45,Z 318.379,A -85,B 0,C 180,E1 -727.386,E2 -727.386} C_VEL
LIN {X 0,Y 601.426,Z 318.383,A -85,B 0,C 180,E1 -730.096,E2 -730.096} C_VEL
LIN {X 0,Y 601.418,Z 318.387,A -85,B 0,C 180,E1 -732.829,E2 -732.829} C_VEL
LIN {X 0,Y 601.408,Z 318.385,A -85,B 0,C 180,E1 -735.592,E2 -735.592} C_VEL
LIN {X 0,Y 601.396,Z 318.39,A -85,B 0,C 180,E1 -737.689,E2 -737.689} C_VEL
LIN {X 0,Y 601.423,Z 318.383,A -85,B 0,C 180,E1 -740.523,E2 -740.523} C_VEL
LIN {X 0,Y 601.42,Z 318.384,A -85,B 0,C 180,E1 -743.411,E2 -743.411} C_VEL
LIN {X 0,Y 601.4,Z 318.387,A -85,B 0,C 180,E1 -746.364,E2 -746.364} C_VEL
LIN {X 0,Y 601.438,Z 318.383,A -85,B 0,C 180,E1 -748.792,E2 -748.792} C_VEL
LIN {X 0,Y 601.412,Z 318.384,A -85,B 0,C 180,E1 -751.456,E2 -751.456} C_VEL
LIN {X 0,Y 601.426,Z 318.382,A -85,B 0,C 180,E1 -754.119,E2 -754.119} C_VEL
LIN {X 0,Y 601.413,Z 318.384,A -85,B 0,C 180,E1 -756.583,E2 -756.583} C_VEL
LIN {X 0,Y 601.435,Z 318.385,A -85,B 0,C 180,E1 -759.537,E2 -759.537} C_VEL
LIN {X 0,Y 601.41,Z 318.384,A -85,B 0,C 180,E1 -762.592,E2 -762.592} C_VEL
LIN {X 0,Y 601.418,Z 318.385,A -85,B 0,C 180,E1 -764.536,E2 -764.536} C_VEL
LIN {X 0,Y 601.403,Z 318.385,A -85,B 0,C 180,E1 -767.331,E2 -767.331} C_VEL
LIN {X 0,Y 601.405,Z 318.385,A -85,B 0,C 180,E1 -770.006,E2 -770.006} C_VEL
LIN {X 0,Y 601.434,Z 318.382,A -85,B 0,C 180,E1 -772.618,E2 -772.618} C_VEL
LIN {X 0,Y 601.44,Z 318.382,A -85,B 0,C 180,E1 -775.071,E2 -775.071} C_VEL
LIN {X 0,Y 601.439,Z 318.475,A -85,B 0,C 180,E1 -777.139,E2 -777.139} C_VEL
LIN {X 0,Y 601.516,Z 325.891,A -85,B 0,C 180,E1 -779.454,E2 -779.454} C_VEL
LIN {X 0,Y 601.484,Z 334.885,A -85,B 0,C 180,E1 -782.137,E2 -782.137} C_VEL
LIN {X 0,Y 601.435,Z 343.826,A -85,B 0,C 180,E1 -784.754,E2 -784.754} C_VEL
LIN {X 0,Y 601.411,Z 353.041,A -85,B 0,C 180,E1 -787.396,E2 -787.396} C_VEL
LIN {X 0,Y 601.416,Z 362.986,A -85,B 0,C 180,E1 -790.192,E2 -790.192} C_VEL
LIN {X 0,Y 601.367,Z 373.205,A -85,B 0,C 180,E1 -793.013,E2 -793.013} C_VEL
LIN {X 0,Y 601.396,Z 382.146,A -85,B 0,C 180,E1 -795.449,E2 -795.449} C_VEL
LIN {X 0,Y 601.367,Z 392.365,A -85,B 0,C 180,E1 -798.2,E2 -798.2} C_VEL
LIN {X 0,Y 601.339,Z 401.306,A -85,B 0,C 180,E1 -800.584,E2 -800.584} C_VEL
LIN {X 0,Y 601.503,Z 414.507,A -85,B 0,C 180,E1 -800.926,E2 -800.926} C_VEL
LIN {X 0,Y 601.447,Z 423.558,A -85,B 0,C 180,E1 -801.264,E2 -801.264} C_VEL
LIN {X 0,Y 601.426,Z 432.252,A -85,B 0,C 180,E1 -801.686,E2 -801.686} C_VEL
LIN {X 0,Y 601.41,Z 440.557,A -85,B 0,C 180,E1 -802.193,E2 -802.193} C_VEL
LIN {X 0,Y 601.413,Z 448.412,A -85,B 0,C 180,E1 -802.784,E2 -802.784} C_VEL
LIN {X 0,Y 601.411,Z 455.604,A -85,B 0,C 180,E1 -803.444,E2 -803.444} C_VEL
LIN {X 0,Y 601.391,Z 463.198,A -85,B 0,C 180,E1 -804.3,E2 -804.3} C_VEL
LIN {X 0,Y 601.38,Z 469.033,A -85,B 0,C 180,E1 -805.141,E2 -805.141} C_VEL
LIN {X 0,Y 601.345,Z 473.635,A -85,B 0,C 180,E1 -805.98,E2 -805.98} C_VEL
LIN {X 0,Y 601.343,Z 476.625,A -85,B 0,C 180,E1 -806.651,E2 -806.651} C_VEL
LIN {X 0,Y 601.326,Z 478.935,A -85,B 0,C 180,E1 -807.321,E2 -807.321} C_VEL
LIN {X 0,Y 601.343,Z 480.681,A -85,B 0,C 180,E1 -807.992,E2 -807.992} C_VEL
LIN {X 0,Y 601.345,Z 481.935,A -85,B 0,C 180,E1 -808.662,E2 -808.662} C_VEL
LIN {X 0,Y 601.335,Z 482.714,A -85,B 0,C 180,E1 -809.331,E2 -809.331} C_VEL
LIN {X 0,Y 601.332,Z 483,A -85,B 0,C 180,E1 -810.001,E2 -810.001} C_VEL
LIN {X 0,Y 601.335,Z 482.713,A -85,B 0,C 180,E1 -810.671,E2 -810.671} C_VEL
LIN {X 0,Y 601.345,Z 481.933,A -85,B 0,C 180,E1 -811.34,E2 -811.34} C_VEL
LIN {X 0,Y 601.343,Z 480.677,A -85,B 0,C 180,E1 -812.01,E2 -812.01} C_VEL
LIN {X 0,Y 601.342,Z 477.783,A -85,B 0,C 180,E1 -813.016,E2 -813.016} C_VEL
LIN {X 0,Y 601.364,Z 475.143,A -85,B 0,C 180,E1 -813.686,E2 -813.686} C_VEL
LIN {X 0,Y 601.341,Z 469.98,A -85,B 0,C 180,E1 -814.693,E2 -814.693} C_VEL
LIN {X 0,Y 601.383,Z 464.424,A -85,B 0,C 180,E1 -815.533,E2 -815.533} C_VEL
LIN {X 0,Y 601.394,Z 457.154,A -85,B 0,C 180,E1 -816.403,E2 -816.403} C_VEL
LIN {X 0,Y 601.417,Z 449.406,A -85,B 0,C 180,E1 -817.133,E2 -817.133} C_VEL
LIN {X 0,Y 601.432,Z 441.75,A -85,B 0,C 180,E1 -817.724,E2 -817.724} C_VEL
LIN {X 0,Y 601.437,Z 433.708,A -85,B 0,C 180,E1 -818.231,E2 -818.231} C_VEL
LIN {X 0,Y 601.458,Z 425.374,A -85,B 0,C 180,E1 -818.653,E2 -818.653} C_VEL
LIN {X 0,Y 601.468,Z 416.867,A -85,B 0,C 180,E1 -818.992,E2 -818.992} C_VEL
LIN {X 0,Y 601.503,Z 407.553,A -85,B 0,C 180,E1 -819.267,E2 -819.267} C_VEL
LIN {X 0,Y 601.341,Z 401.299,A -85,B 0,C 180,E1 -819.418,E2 -819.418} C_VEL
LIN {X 0,Y 601.364,Z 391.081,A -85,B 0,C 180,E1 -822.144,E2 -822.144} C_VEL
LIN {X 0,Y 601.363,Z 380.862,A -85,B 0,C 180,E1 -824.899,E2 -824.899} C_VEL
LIN {X 0,Y 601.404,Z 370.643,A -85,B 0,C 180,E1 -827.689,E2 -827.689} C_VEL
LIN {X 0,Y 601.416,Z 360.425,A -85,B 0,C 180,E1 -830.523,E2 -830.523} C_VEL
LIN {X 0,Y 601.404,Z 351.483,A -85,B 0,C 180,E1 -833.047,E2 -833.047} C_VEL
LIN {X 0,Y 601.47,Z 341.643,A -85,B 0,C 180,E1 -835.878,E2 -835.878} C_VEL
LIN {X 0,Y 601.452,Z 331.71,A -85,B 0,C 180,E1 -838.791,E2 -838.791} C_VEL
LIN {X 0,Y 601.531,Z 322.868,A -85,B 0,C 180,E1 -841.472,E2 -841.472} C_VEL
LIN {X 0,Y 601.424,Z 318.384,A -85,B 0,C 180,E1 -842.903,E2 -842.903} C_VEL
LIN {X 0,Y 601.391,Z 318.39,A -85,B 0,C 180,E1 -845.755,E2 -845.755} C_VEL
LIN {X 0,Y 601.418,Z 318.384,A -85,B 0,C 180,E1 -848.469,E2 -848.469} C_VEL
LIN {X 0,Y 601.417,Z 318.384,A -85,B 0,C 180,E1 -850.875,E2 -850.875} C_VEL
LIN {X 0,Y 601.456,Z 318.379,A -85,B 0,C 180,E1 -853.584,E2 -853.584} C_VEL
LIN {X 0,Y 601.433,Z 318.385,A -85,B 0,C 180,E1 -856.428,E2 -856.428} C_VEL
LIN {X 0,Y 601.421,Z 318.383,A -85,B 0,C 180,E1 -859.427,E2 -859.427} C_VEL
LIN {X 0,Y 601.409,Z 318.384,A -85,B 0,C 180,E1 -861.731,E2 -861.731} C_VEL
LIN {X 0,Y 601.387,Z 318.387,A -85,B 0,C 180,E1 -864.245,E2 -864.245} C_VEL
LIN {X 0,Y 601.415,Z 318.384,A -85,B 0,C 180,E1 -866.685,E2 -866.685} C_VEL
LIN {X 0,Y 601.41,Z 318.385,A -85,B 0,C 180,E1 -869.057,E2 -869.057} C_VEL
LIN {X 0,Y 601.434,Z 318.382,A -85,B 0,C 180,E1 -871.373,E2 -871.373} C_VEL
LIN {X 0,Y 601.4,Z 318.386,A -85,B 0,C 180,E1 -873.636,E2 -873.636} C_VEL
LIN {X 0,Y 601.418,Z 318.386,A -85,B 0,C 180,E1 -876.589,E2 -876.589} C_VEL
LIN {X 0,Y 601.422,Z 318.383,A -85,B 0,C 180,E1 -879.477,E2 -879.477} C_VEL
LIN {X 0,Y 601.395,Z 318.389,A -85,B 0,C 180,E1 -882.311,E2 -882.311} C_VEL
LIN {X 0,Y 601.41,Z 318.385,A -85,B 0,C 180,E1 -884.408,E2 -884.408} C_VEL
LIN {X 0,Y 601.417,Z 318.386,A -85,B 0,C 180,E1 -887.171,E2 -887.171} C_VEL
LIN {X 0,Y 601.425,Z 318.383,A -85,B 0,C 180,E1 -889.904,E2 -889.904} C_VEL
LIN {X 0,Y 601.447,Z 318.38,A -85,B 0,C 180,E1 -892.614,E2 -892.614} C_VEL
LIN {X 0,Y 601.427,Z 318.386,A -85,B 0,C 180,E1 -895.307,E2 -895.307} C_VEL
LIN {X 0,Y 601.424,Z 318.383,A -85,B 0,C 180,E1 -897.99,E2 -897.99} C_VEL
LIN {X 0,Y 601.454,Z 318.379,A -85,B 0,C 180,E1 -900.669,E2 -900.669} C_VEL
LIN {X 0,Y 601.422,Z 318.384,A -85,B 0,C 180,E1 -903.349,E2 -903.349} C_VEL
LIN {X 0,Y 601.42,Z 318.386,A -85,B 0,C 180,E1 -906.036,E2 -906.036} C_VEL
LIN {X 0,Y 601.411,Z 318.384,A -85,B 0,C 180,E1 -908.737,E2 -908.737} C_VEL
LIN {X 0,Y 601.414,Z 318.384,A -85,B 0,C 180,E1 -911.458,E2 -911.458} C_VEL
LIN {X 0,Y 601.412,Z 318.384,A -85,B 0,C 180,E1 -912.373,E2 -912.373} C_VEL
LIN {X 0,Y 600.744,Z 318.47,A -85,B 0,C 180,E1 -912.932,E2 -912.932} C_VEL
LIN {X 0,Y 597.892,Z 318.823,A -85,B 0,C 180,E1 -913.84,E2 -913.84} C_VEL
LIN {X 0,Y 595.482,Z 319.124,A -85,B 0,C 180,E1 -914.57,E2 -914.57} C_VEL
LIN {X 0,Y 594.445,Z 319.253,A -85,B 0,C 180,E1 -915.134,E2 -915.134} C_VEL
LIN {X 0,Y 594.36,Z 319.262,A -85,B 0,C 180,E1 -915.325,E2 -915.325} C_VEL
LIN {X 0,Y 594.383,Z 319.26,A -85,B 0,C 180,E1 -917.193,E2 -917.193} C_VEL
LIN {X 0,Y 594.311,Z 319.272,A -85,B 0,C 180,E1 -917.905,E2 -917.905} C_VEL
LIN {X 0,Y 594.301,Z 323.411,A -85,B 0,C 180,E1 -920.778,E2 -920.778} C_VEL
LIN {X 0,Y 594.293,Z 326.568,A -85,B 0,C 180,E1 -922.969,E2 -922.969} C_VEL
LIN {X 0,Y 594.253,Z 329.86,A -85,B 0,C 180,E1 -925.198,E2 -925.198} C_VEL
LIN {X 0,Y 594.249,Z 333.435,A -85,B 0,C 180,E1 -927.5,E2 -927.5} C_VEL
LIN {X 0,Y 594.24,Z 337.868,A -85,B 0,C 180,E1 -930.303,E2 -930.303} C_VEL
LIN {X 0,Y 594.239,Z 342.139,A -85,B 0,C 180,E1 -932.958,E2 -932.958} C_VEL
LIN {X 0,Y 594.205,Z 346.152,A -85,B 0,C 180,E1 -935.418,E2 -935.418} C_VEL
LIN {X 0,Y 594.199,Z 350.336,A -85,B 0,C 180,E1 -937.953,E2 -937.953} C_VEL
LIN {X 0,Y 594.238,Z 354.703,A -85,B 0,C 180,E1 -940.576,E2 -940.576} C_VEL
LIN {X 0,Y 594.487,Z 360.343,A -85,B 0,C 180,E1 -940.74,E2 -940.74} C_VEL
LIN {X 0,Y 594.459,Z 372.268,A -85,B 0,C 180,E1 -941.146,E2 -941.146} C_VEL
LIN {X 0,Y 594.403,Z 382.667,A -85,B 0,C 180,E1 -941.656,E2 -941.656} C_VEL
LIN {X 0,Y 594.355,Z 390.754,A -85,B 0,C 180,E1 -942.159,E2 -942.159} C_VEL
LIN {X 0,Y 594.358,Z 398.696,A -85,B 0,C 180,E1 -942.767,E2 -942.767} C_VEL
LIN {X 0,Y 594.333,Z 405.836,A -85,B 0,C 180,E1 -943.434,E2 -943.434} C_VEL
LIN {X 0,Y 594.303,Z 412.914,A -85,B 0,C 180,E1 -944.242,E2 -944.242} C_VEL
LIN {X 0,Y 594.306,Z 419.414,A -85,B 0,C 180,E1 -945.195,E2 -945.195} C_VEL
LIN {X 0,Y 594.278,Z 422.555,A -85,B 0,C 180,E1 -945.753,E2 -945.753} C_VEL
LIN {X 0,Y 594.264,Z 426.753,A -85,B 0,C 180,E1 -946.691,E2 -946.691} C_VEL
LIN {X 0,Y 594.27,Z 429.741,A -85,B 0,C 180,E1 -947.615,E2 -947.615} C_VEL
LIN {X 0,Y 594.214,Z 431.7,A -85,B 0,C 180,E1 -948.521,E2 -948.521} C_VEL
LIN {X 0,Y 594.236,Z 432.738,A -85,B 0,C 180,E1 -949.421,E2 -949.421} C_VEL
LIN {X 0,Y 594.199,Z 432.905,A -85,B 0,C 180,E1 -950.305,E2 -950.305} C_VEL
LIN {X 0,Y 594.205,Z 432.053,A -85,B 0,C 180,E1 -951.315,E2 -951.315} C_VEL
LIN {X 0,Y 594.232,Z 429.898,A -85,B 0,C 180,E1 -952.409,E2 -952.409} C_VEL
LIN {X 0,Y 594.253,Z 426.228,A -85,B 0,C 180,E1 -953.532,E2 -953.532} C_VEL
LIN {X 0,Y 594.269,Z 422.334,A -85,B 0,C 180,E1 -954.377,E2 -954.377} C_VEL
LIN {X 0,Y 594.301,Z 417.272,A -85,B 0,C 180,E1 -955.233,E2 -955.233} C_VEL
LIN {X 0,Y 594.307,Z 411.215,A -85,B 0,C 180,E1 -956.052,E2 -956.052} C_VEL
LIN {X 0,Y 594.339,Z 404.969,A -85,B 0,C 180,E1 -956.743,E2 -956.743} C_VEL
LIN {X 0,Y 594.364,Z 398.238,A -85,B 0,C 180,E1 -957.362,E2 -957.362} C_VEL
LIN {X 0,Y 594.376,Z 389.846,A -85,B 0,C 180,E1 -957.995,E2 -957.995} C_VEL
LIN {X 0,Y 594.386,Z 380.157,A -85,B 0,C 180,E1 -958.577,E2 -958.577} C_VEL
LIN {X 0,Y 594.434,Z 369.555,A -85,B 0,C 180,E1 -959.049,E2 -959.049} C_VEL
LIN {X 0,Y 594.488,Z 359.023,A -85,B 0,C 180,E1 -959.384,E2 -959.384} C_VEL
LIN {X 0,Y 594.25,Z 354.708,A -85,B 0,C 180,E1 -959.51,E2 -959.51} C_VEL
LIN {X 0,Y 594.254,Z 349.678,A -85,B 0,C 180,E1 -962.532,E2 -962.532} C_VEL
LIN {X 0,Y 594.264,Z 344.648,A -85,B 0,C 180,E1 -965.59,E2 -965.59} C_VEL
LIN {X 0,Y 594.25,Z 341.12,A -85,B 0,C 180,E1 -967.761,E2 -967.761} C_VEL
LIN {X 0,Y 594.227,Z 337.624,A -85,B 0,C 180,E1 -969.94,E2 -969.94} C_VEL
LIN {X 0,Y 594.214,Z 334.221,A -85,B 0,C 180,E1 -972.09,E2 -972.09} C_VEL
LIN {X 0,Y 594.224,Z 330.907,A -85,B 0,C 180,E1 -974.214,E2 -974.214} C_VEL
LIN {X 0,Y 594.218,Z 327.734,A -85,B 0,C 180,E1 -976.316,E2 -976.316} C_VEL
LIN {X 0,Y 594.344,Z 323.651,A -85,B 0,C 180,E1 -979.093,E2 -979.093} C_VEL
LIN {X 0,Y 594.306,Z 319.628,A -85,B 0,C 180,E1 -981.841,E2 -981.841} C_VEL
LIN {X 0,Y 594.399,Z 319.259,A -85,B 0,C 180,E1 -983.299,E2 -983.299} C_VEL
LIN {X 0,Y 594.359,Z 319.266,A -85,B 0,C 180,E1 -985.931,E2 -985.931} C_VEL
LIN {X 0,Y 594.382,Z 319.26,A -85,B 0,C 180,E1 -987.966,E2 -987.966} C_VEL
LIN {X 0,Y 594.417,Z 319.257,A -85,B 0,C 180,E1 -990.677,E2 -990.677} C_VEL
LIN {X 0,Y 594.381,Z 319.262,A -85,B 0,C 180,E1 -993.388,E2 -993.388} C_VEL
LIN {X 0,Y 594.362,Z 319.262,A -85,B 0,C 180,E1 -996.108,E2 -996.108} C_VEL
LIN {X 0,Y 594.396,Z 319.258,A -85,B 0,C 180,E1 -998.841,E2 -998.841} C_VEL
LIN {X 0,Y 594.385,Z 319.261,A -85,B 0,C 180,E1 -1001.595,E2 -1001.595} C_VEL
LIN {X 0,Y 594.379,Z 319.261,A -85,B 0,C 180,E1 -1004.376,E2 -1004.376} C_VEL
LIN {X 0,Y 594.381,Z 319.26,A -85,B 0,C 180,E1 -1007.193,E2 -1007.193} C_VEL
LIN {X 0,Y 594.37,Z 319.263,A -85,B 0,C 180,E1 -1010.053,E2 -1010.053} C_VEL
LIN {X 0,Y 594.353,Z 319.264,A -85,B 0,C 180,E1 -1012.967,E2 -1012.967} C_VEL
LIN {X 0,Y 594.367,Z 319.264,A -85,B 0,C 180,E1 -1015.192,E2 -1015.192} C_VEL
LIN {X 0,Y 594.37,Z 319.265,A -85,B 0,C 180,E1 -1017.526,E2 -1017.526} C_VEL
LIN {X 0,Y 594.388,Z 319.259,A -85,B 0,C 180,E1 -1020.331,E2 -1020.331} C_VEL
LIN {X 0,Y 594.369,Z 319.261,A -85,B 0,C 180,E1 -1022.949,E2 -1022.949} C_VEL
LIN {X 0,Y 594.372,Z 319.261,A -85,B 0,C 180,E1 -1025.406,E2 -1025.406} C_VEL
LIN {X 0,Y 594.375,Z 319.26,A -85,B 0,C 180,E1 -1027.94,E2 -1027.94} C_VEL
LIN {X 0,Y 594.376,Z 319.263,A -85,B 0,C 180,E1 -1030.824,E2 -1030.824} C_VEL
LIN {X 0,Y 594.372,Z 319.265,A -85,B 0,C 180,E1 -1033.297,E2 -1033.297} C_VEL
LIN {X 0,Y 594.368,Z 319.262,A -85,B 0,C 180,E1 -1036.159,E2 -1036.159} C_VEL
LIN {X 0,Y 594.373,Z 319.262,A -85,B 0,C 180,E1 -1039.177,E2 -1039.177} C_VEL
LIN {X 0,Y 594.382,Z 319.261,A -85,B 0,C 180,E1 -1042.06,E2 -1042.06} C_VEL
LIN {X 0,Y 594.372,Z 319.261,A -85,B 0,C 180,E1 -1044.671,E2 -1044.671} C_VEL
LIN {X 0,Y 594.366,Z 319.262,A -85,B 0,C 180,E1 -1047.088,E2 -1047.088} C_VEL
LIN {X 0,Y 594.388,Z 319.258,A -85,B 0,C 180,E1 -1049.669,E2 -1049.669} C_VEL
LIN {X 0,Y 594.377,Z 319.262,A -85,B 0,C 180,E1 -1052.54,E2 -1052.54} C_VEL
LIN {X 0,Y 594.365,Z 319.262,A -85,B 0,C 180,E1 -1054.807,E2 -1054.807} C_VEL
LIN {X 0,Y 594.391,Z 319.259,A -85,B 0,C 180,E1 -1057.255,E2 -1057.255} C_VEL
LIN {X 0,Y 594.367,Z 319.264,A -85,B 0,C 180,E1 -1059.947,E2 -1059.947} C_VEL
LIN {X 0,Y 594.38,Z 319.26,A -85,B 0,C 180,E1 -1062.807,E2 -1062.807} C_VEL
LIN {X 0,Y 594.378,Z 319.261,A -85,B 0,C 180,E1 -1065.826,E2 -1065.826} C_VEL
LIN {X 0,Y 594.385,Z 319.262,A -85,B 0,C 180,E1 -1068.405,E2 -1068.405} C_VEL
LIN {X 0,Y 594.394,Z 319.26,A -85,B 0,C 180,E1 -1071.159,E2 -1071.159} C_VEL
LIN {X 0,Y 594.361,Z 319.262,A -85,B 0,C 180,E1 -1073.892,E2 -1073.892} C_VEL
LIN {X 0,Y 594.371,Z 319.261,A -85,B 0,C 180,E1 -1076.611,E2 -1076.611} C_VEL
LIN {X 0,Y 594.417,Z 319.257,A -85,B 0,C 180,E1 -1079.323,E2 -1079.323} C_VEL
LIN {X 0,Y 594.397,Z 319.26,A -85,B 0,C 180,E1 -1082.033,E2 -1082.033} C_VEL
LIN {X 0,Y 594.386,Z 319.259,A -85,B 0,C 180,E1 -1084.748,E2 -1084.748} C_VEL
LIN {X 0,Y 594.413,Z 319.256,A -85,B 0,C 180,E1 -1087.474,E2 -1087.474} C_VEL
LIN {X 0,Y 594.387,Z 319.261,A -85,B 0,C 180,E1 -1090.217,E2 -1090.217} C_VEL
LIN {X 0,Y 594.367,Z 319.264,A -85,B 0,C 180,E1 -1092.984,E2 -1092.984} C_VEL
LIN {X 0,Y 594.361,Z 319.262,A -85,B 0,C 180,E1 -1095.782,E2 -1095.782} C_VEL
LIN {X 0,Y 594.377,Z 319.261,A -85,B 0,C 180,E1 -1098.618,E2 -1098.618} C_VEL
LIN {X 0,Y 594.36,Z 319.264,A -85,B 0,C 180,E1 -1101.504,E2 -1101.504} C_VEL
LIN {X 0,Y 594.379,Z 319.26,A -85,B 0,C 180,E1 -1104.447,E2 -1104.447} C_VEL
LIN {X 0,Y 594.385,Z 319.259,A -85,B 0,C 180,E1 -1106.7,E2 -1106.7} C_VEL
LIN {X 0,Y 594.381,Z 319.26,A -85,B 0,C 180,E1 -1108.999,E2 -1108.999} C_VEL
LIN {X 0,Y 594.371,Z 319.261,A -85,B 0,C 180,E1 -1111.644,E2 -1111.644} C_VEL
LIN {X 0,Y 594.394,Z 319.261,A -85,B 0,C 180,E1 -1114.579,E2 -1114.579} C_VEL
LIN {X 0,Y 594.382,Z 319.263,A -85,B 0,C 180,E1 -1117.087,E2 -1117.087} C_VEL
LIN {X 0,Y 594.369,Z 319.262,A -85,B 0,C 180,E1 -1119.776,E2 -1119.776} C_VEL
LIN {X 0,Y 594.366,Z 319.262,A -85,B 0,C 180,E1 -1122.376,E2 -1122.376} C_VEL
LIN {X 0,Y 594.357,Z 319.263,A -85,B 0,C 180,E1 -1125.192,E2 -1125.192} C_VEL
LIN {X 0,Y 594.362,Z 319.262,A -85,B 0,C 180,E1 -1127.626,E2 -1127.626} C_VEL
LIN {X 0,Y 594.386,Z 319.262,A -85,B 0,C 180,E1 -1130.322,E2 -1130.322} C_VEL
LIN {X 0,Y 594.382,Z 319.263,A -85,B 0,C 180,E1 -1132.915,E2 -1132.915} C_VEL
LIN {X 0,Y 594.381,Z 319.26,A -85,B 0,C 180,E1 -1135.862,E2 -1135.862} C_VEL
LIN {X 0,Y 594.381,Z 319.277,A -85,B 0,C 180,E1 -1136.95,E2 -1136.95} C_VEL
LIN {X 0,Y 594.574,Z 324.625,A -85,B 0,C 180,E1 -1138.663,E2 -1138.663} C_VEL
LIN {X 0,Y 594.45,Z 333.536,A -85,B 0,C 180,E1 -1141.405,E2 -1141.405} C_VEL
LIN {X 0,Y 594.467,Z 343.826,A -85,B 0,C 180,E1 -1144.437,E2 -1144.437} C_VEL
LIN {X 0,Y 594.365,Z 353.571,A -85,B 0,C 180,E1 -1147.265,E2 -1147.265} C_VEL
LIN {X 0,Y 594.388,Z 362.986,A -85,B 0,C 180,E1 -1149.948,E2 -1149.948} C_VEL
LIN {X 0,Y 594.31,Z 373.205,A -85,B 0,C 180,E1 -1152.805,E2 -1152.805} C_VEL
LIN {X 0,Y 594.315,Z 383.423,A -85,B 0,C 180,E1 -1155.622,E2 -1155.622} C_VEL
LIN {X 0,Y 594.296,Z 393.642,A -85,B 0,C 180,E1 -1158.403,E2 -1158.403} C_VEL
LIN {X 0,Y 594.264,Z 401.306,A -85,B 0,C 180,E1 -1160.471,E2 -1160.471} C_VEL
LIN {X 0,Y 594.503,Z 410.112,A -85,B 0,C 180,E1 -1160.689,E2 -1160.689} C_VEL
LIN {X 0,Y 594.439,Z 421.638,A -85,B 0,C 180,E1 -1161.074,E2 -1161.074} C_VEL
LIN {X 0,Y 594.401,Z 432.254,A -85,B 0,C 180,E1 -1161.587,E2 -1161.587} C_VEL
LIN {X 0,Y 594.368,Z 440.559,A -85,B 0,C 180,E1 -1162.1,E2 -1162.1} C_VEL
LIN {X 0,Y 594.354,Z 448.413,A -85,B 0,C 180,E1 -1162.698,E2 -1162.698} C_VEL
LIN {X 0,Y 594.342,Z 455.522,A -85,B 0,C 180,E1 -1163.357,E2 -1163.357} C_VEL
LIN {X 0,Y 594.318,Z 463.198,A -85,B 0,C 180,E1 -1164.232,E2 -1164.232} C_VEL
LIN {X 0,Y 594.289,Z 469.033,A -85,B 0,C 180,E1 -1165.082,E2 -1165.082} C_VEL
LIN {X 0,Y 594.261,Z 473.635,A -85,B 0,C 180,E1 -1165.932,E2 -1165.932} C_VEL
LIN {X 0,Y 594.265,Z 476.625,A -85,B 0,C 180,E1 -1166.611,E2 -1166.611} C_VEL
LIN {X 0,Y 594.228,Z 478.935,A -85,B 0,C 180,E1 -1167.289,E2 -1167.289} C_VEL
LIN {X 0,Y 594.242,Z 480.681,A -85,B 0,C 180,E1 -1167.968,E2 -1167.968} C_VEL
LIN {X 0,Y 594.245,Z 481.936,A -85,B 0,C 180,E1 -1168.646,E2 -1168.646} C_VEL
LIN {X 0,Y 594.235,Z 482.713,A -85,B 0,C 180,E1 -1169.323,E2 -1169.323} C_VEL
LIN {X 0,Y 594.233,Z 483,A -85,B 0,C 180,E1 -1170.001,E2 -1170.001} C_VEL
LIN {X 0,Y 594.235,Z 482.712,A -85,B 0,C 180,E1 -1170.679,E2 -1170.679} C_VEL
LIN {X 0,Y 594.245,Z 481.934,A -85,B 0,C 180,E1 -1171.356,E2 -1171.356} C_VEL
LIN {X 0,Y 594.242,Z 480.677,A -85,B 0,C 180,E1 -1172.034,E2 -1172.034} C_VEL
LIN {X 0,Y 594.245,Z 477.784,A -85,B 0,C 180,E1 -1173.052,E2 -1173.052} C_VEL
LIN {X 0,Y 594.285,Z 475.143,A -85,B 0,C 180,E1 -1173.73,E2 -1173.73} C_VEL
LIN {X 0,Y 594.256,Z 469.98,A -85,B 0,C 180,E1 -1174.75,E2 -1174.75} C_VEL
LIN {X 0,Y 594.318,Z 463.183,A -85,B 0,C 180,E1 -1175.77,E2 -1175.77} C_VEL
LIN {X 0,Y 594.343,Z 455.51,A -85,B 0,C 180,E1 -1176.644,E2 -1176.644} C_VEL
LIN {X 0,Y 594.355,Z 448.394,A -85,B 0,C 180,E1 -1177.304,E2 -1177.304} C_VEL
LIN {X 0,Y 594.373,Z 440.535,A -85,B 0,C 180,E1 -1177.901,E2 -1177.901} C_VEL
LIN {X 0,Y 594.421,Z 430.723,A -85,B 0,C 180,E1 -1178.5,E2 -1178.5} C_VEL
LIN {X 0,Y 594.464,Z 419.275,A -85,B 0,C 180,E1 -1179.013,E2 -1179.013} C_VEL
LIN {X 0,Y 594.505,Z 410.044,A -85,B 0,C 180,E1 -1179.313,E2 -1179.313} C_VEL
LIN {X 0,Y 594.265,Z 401.299,A -85,B 0,C 180,E1 -1179.531,E2 -1179.531} C_VEL
LIN {X 0,Y 594.3,Z 391.081,A -85,B 0,C 180,E1 -1182.291,E2 -1182.291} C_VEL
LIN {X 0,Y 594.297,Z 380.862,A -85,B 0,C 180,E1 -1185.081,E2 -1185.081} C_VEL
LIN {X 0,Y 594.365,Z 370.643,A -85,B 0,C 180,E1 -1187.905,E2 -1187.905} C_VEL
LIN {X 0,Y 594.37,Z 360.425,A -85,B 0,C 180,E1 -1190.778,E2 -1190.778} C_VEL
LIN {X 0,Y 594.413,Z 351.483,A -85,B 0,C 180,E1 -1193.334,E2 -1193.334} C_VEL
LIN {X 0,Y 594.444,Z 341.238,A -85,B 0,C 180,E1 -1196.327,E2 -1196.327} C_VEL
LIN {X 0,Y 594.454,Z 332.139,A -85,B 0,C 180,E1 -1198.995,E2 -1198.995} C_VEL
LIN {X 0,Y 594.55,Z 323.531,A -85,B 0,C 180,E1 -1201.669,E2 -1201.669} C_VEL
LIN {X 0,Y 594.389,Z 319.262,A -85,B 0,C 180,E1 -1203.051,E2 -1203.051} C_VEL
LIN {X 0,Y 594.355,Z 319.264,A -85,B 0,C 180,E1 -1205.409,E2 -1205.409} C_VEL
LIN {X 0,Y 594.39,Z 319.26,A -85,B 0,C 180,E1 -1207.941,E2 -1207.941} C_VEL
LIN {X 0,Y 594.379,Z 319.262,A -85,B 0,C 180,E1 -1210.822,E2 -1210.822} C_VEL
LIN {X 0,Y 594.381,Z 319.262,A -85,B 0,C 180,E1 -1213.84,E2 -1213.84} C_VEL
LIN {X 0,Y 594.371,Z 319.262,A -85,B 0,C 180,E1 -1216.701,E2 -1216.701} C_VEL
LIN {X 0,Y 594.376,Z 319.261,A -85,B 0,C 180,E1 -1219.433,E2 -1219.433} C_VEL
LIN {X 0,Y 594.391,Z 319.262,A -85,B 0,C 180,E1 -1222.392,E2 -1222.392} C_VEL
LIN {X 0,Y 594.383,Z 319.26,A -85,B 0,C 180,E1 -1225.42,E2 -1225.42} C_VEL
LIN {X 0,Y 594.38,Z 319.262,A -85,B 0,C 180,E1 -1228.358,E2 -1228.358} C_VEL
LIN {X 0,Y 594.388,Z 319.259,A -85,B 0,C 180,E1 -1231.042,E2 -1231.042} C_VEL
LIN {X 0,Y 594.386,Z 319.261,A -85,B 0,C 180,E1 -1233.978,E2 -1233.978} C_VEL
LIN {X 0,Y 594.385,Z 319.261,A -85,B 0,C 180,E1 -1236.295,E2 -1236.295} C_VEL
LIN {X 0,Y 594.397,Z 319.258,A -85,B 0,C 180,E1 -1239.224,E2 -1239.224} C_VEL
LIN {X 0,Y 594.347,Z 319.265,A -85,B 0,C 180,E1 -1242.094,E2 -1242.094} C_VEL
LIN {X 0,Y 594.364,Z 319.262,A -85,B 0,C 180,E1 -1244.218,E2 -1244.218} C_VEL
LIN {X 0,Y 594.389,Z 319.259,A -85,B 0,C 180,E1 -1246.321,E2 -1246.321} C_VEL
LIN {X 0,Y 594.38,Z 319.26,A -85,B 0,C 180,E1 -1249.094,E2 -1249.094} C_VEL
LIN {X 0,Y 594.385,Z 319.263,A -85,B 0,C 180,E1 -1251.842,E2 -1251.842} C_VEL
LIN {X 0,Y 594.398,Z 319.258,A -85,B 0,C 180,E1 -1254.572,E2 -1254.572} C_VEL
LIN {X 0,Y 594.4,Z 319.258,A -85,B 0,C 180,E1 -1257.289,E2 -1257.289} C_VEL
LIN {X 0,Y 594.416,Z 319.259,A -85,B 0,C 180,E1 -1259.999,E2 -1259.999} C_VEL
LIN {X 0,Y 594.408,Z 319.257,A -85,B 0,C 180,E1 -1262.71,E2 -1262.71} C_VEL
LIN {X 0,Y 594.385,Z 319.259,A -85,B 0,C 180,E1 -1265.427,E2 -1265.427} C_VEL
LIN {X 0,Y 594.389,Z 319.259,A -85,B 0,C 180,E1 -1267.472,E2 -1267.472} C_VEL
LIN {X 0,Y 594.395,Z 319.258,A -85,B 0,C 180,E1 -1270.215,E2 -1270.215} C_VEL
LIN {X 0,Y 594.367,Z 319.265,A -85,B 0,C 180,E1 -1272.982,E2 -1272.982} C_VEL
LIN {X 0,Y 594.36,Z 319.262,A -85,B 0,C 180,E1 -1275.325,E2 -1275.325} C_VEL
LIN {X 0,Y 593.681,Z 319.375,A -85,B 0,C 180,E1 -1275.892,E2 -1275.892} C_VEL
LIN {X 0,Y 590.789,Z 319.709,A -85,B 0,C 180,E1 -1276.811,E2 -1276.811} C_VEL
LIN {X 0,Y 588.354,Z 320.013,A -85,B 0,C 180,E1 -1277.549,E2 -1277.549} C_VEL
LIN {X 0,Y 587.311,Z 320.246,A -85,B 0,C 180,E1 -1278.117,E2 -1278.117} C_VEL
LIN {X 0,Y 587.228,Z 320.461,A -85,B 0,C 180,E1 -1278.308,E2 -1278.308} C_VEL
LIN {X 0,Y 587.241,Z 324.457,A -85,B 0,C 180,E1 -1281.04,E2 -1281.04} C_VEL
LIN {X 0,Y 587.227,Z 327.627,A -85,B 0,C 180,E1 -1283.262,E2 -1283.262} C_VEL
LIN {X 0,Y 587.186,Z 332.005,A -85,B 0,C 180,E1 -1286.285,E2 -1286.285} C_VEL
LIN {X 0,Y 587.151,Z 336.822,A -85,B 0,C 180,E1 -1289.389,E2 -1289.389} C_VEL
LIN {X 0,Y 587.129,Z 340.634,A -85,B 0,C 180,E1 -1291.801,E2 -1291.801} C_VEL
LIN {X 0,Y 587.118,Z 344.661,A -85,B 0,C 180,E1 -1294.314,E2 -1294.314} C_VEL
LIN {X 0,Y 587.111,Z 348.633,A -85,B 0,C 180,E1 -1296.763,E2 -1296.763} C_VEL
LIN {X 0,Y 587.108,Z 352.917,A -85,B 0,C 180,E1 -1299.377,E2 -1299.377} C_VEL
LIN {X 0,Y 587.149,Z 354.786,A -85,B 0,C 180,E1 -1300.478,E2 -1300.478} C_VEL
LIN {X 0,Y 587.482,Z 361.621,A -85,B 0,C 180,E1 -1300.661,E2 -1300.661} C_VEL
LIN {X 0,Y 587.431,Z 373.261,A -85,B 0,C 180,E1 -1301.085,E2 -1301.085} C_VEL
LIN {X 0,Y 587.391,Z 381.591,A -85,B 0,C 180,E1 -1301.493,E2 -1301.493} C_VEL
LIN {X 0,Y 587.31,Z 389.281,A -85,B 0,C 180,E1 -1301.959,E2 -1301.959} C_VEL
LIN {X 0,Y 587.298,Z 397.052,A -85,B 0,C 180,E1 -1302.539,E2 -1302.539} C_VEL
LIN {X 0,Y 587.287,Z 403.479,A -85,B 0,C 180,E1 -1303.115,E2 -1303.115} C_VEL
LIN {X 0,Y 587.263,Z 409.282,A -85,B 0,C 180,E1 -1303.731,E2 -1303.731} C_VEL
LIN {X 0,Y 587.221,Z 415.161,A -85,B 0,C 180,E1 -1304.485,E2 -1304.485} C_VEL
LIN {X 0,Y 587.229,Z 420.316,A -85,B 0,C 180,E1 -1305.299,E2 -1305.299} C_VEL
LIN {X 0,Y 587.173,Z 425.115,A -85,B 0,C 180,E1 -1306.263,E2 -1306.263} C_VEL
LIN {X 0,Y 587.167,Z 429.39,A -85,B 0,C 180,E1 -1307.447,E2 -1307.447} C_VEL
LIN {X 0,Y 587.117,Z 432.142,A -85,B 0,C 180,E1 -1308.824,E2 -1308.824} C_VEL
LIN {X 0,Y 587.129,Z 432.996,A -85,B 0,C 180,E1 -1310.002,E2 -1310.002} C_VEL
LIN {X 0,Y 587.108,Z 432.392,A -85,B 0,C 180,E1 -1311.084,E2 -1311.084} C_VEL
LIN {X 0,Y 587.151,Z 430.04,A -85,B 0,C 180,E1 -1312.377,E2 -1312.377} C_VEL
LIN {X 0,Y 587.171,Z 427.182,A -85,B 0,C 180,E1 -1313.314,E2 -1313.314} C_VEL
LIN {X 0,Y 587.18,Z 422.071,A -85,B 0,C 180,E1 -1314.476,E2 -1314.476} C_VEL
LIN {X 0,Y 587.222,Z 417.031,A -85,B 0,C 180,E1 -1315.331,E2 -1315.331} C_VEL
LIN {X 0,Y 587.225,Z 410.727,A -85,B 0,C 180,E1 -1316.184,E2 -1316.184} C_VEL
LIN {X 0,Y 587.279,Z 404.271,A -85,B 0,C 180,E1 -1316.895,E2 -1316.895} C_VEL
LIN {X 0,Y 587.304,Z 396.234,A -85,B 0,C 180,E1 -1317.62,E2 -1317.62} C_VEL
LIN {X 0,Y 587.349,Z 386.166,A -85,B 0,C 180,E1 -1318.332,E2 -1318.332} C_VEL
LIN {X 0,Y 587.367,Z 376.94,A -85,B 0,C 180,E1 -1318.835,E2 -1318.835} C_VEL
LIN {X 0,Y 587.44,Z 369.02,A -85,B 0,C 180,E1 -1319.176,E2 -1319.176} C_VEL
LIN {X 0,Y 587.476,Z 359.599,A -85,B 0,C 180,E1 -1319.482,E2 -1319.482} C_VEL
LIN {X 0,Y 587.16,Z 354.699,A -85,B 0,C 180,E1 -1319.632,E2 -1319.632} C_VEL
LIN {X 0,Y 587.158,Z 350.243,A -85,B 0,C 180,E1 -1322.341,E2 -1322.341} C_VEL
LIN {X 0,Y 587.167,Z 345.536,A -85,B 0,C 180,E1 -1325.232,E2 -1325.232} C_VEL
LIN {X 0,Y 587.158,Z 341.926,A -85,B 0,C 180,E1 -1327.478,E2 -1327.478} C_VEL
LIN {X 0,Y 587.167,Z 338.414,A -85,B 0,C 180,E1 -1329.689,E2 -1329.689} C_VEL
LIN {X 0,Y 587.13,Z 335.004,A -85,B 0,C 180,E1 -1331.866,E2 -1331.866} C_VEL
LIN {X 0,Y 587.148,Z 331.68,A -85,B 0,C 180,E1 -1334.019,E2 -1334.019} C_VEL
LIN {X 0,Y 587.158,Z 327.613,A -85,B 0,C 180,E1 -1336.854,E2 -1336.854} C_VEL
LIN {X 0,Y 587.276,Z 323.443,A -85,B 0,C 180,E1 -1339.658,E2 -1339.658} C_VEL
LIN {X 0,Y 587.239,Z 320.425,A -85,B 0,C 180,E1 -1341.742,E2 -1341.742} C_VEL
LIN {X 0,Y 587.364,Z 320.135,A -85,B 0,C 180,E1 -1343.264,E2 -1343.264} C_VEL
LIN {X 0,Y 587.313,Z 320.143,A -85,B 0,C 180,E1 -1345.882,E2 -1345.882} C_VEL
LIN {X 0,Y 587.353,Z 320.135,A -85,B 0,C 180,E1 -1347.942,E2 -1347.942} C_VEL
LIN {X 0,Y 587.387,Z 320.133,A -85,B 0,C 180,E1 -1350.685,E2 -1350.685} C_VEL
LIN {X 0,Y 587.331,Z 320.14,A -85,B 0,C 180,E1 -1353.429,E2 -1353.429} C_VEL
LIN {X 0,Y 587.354,Z 320.136,A -85,B 0,C 180,E1 -1355.492,E2 -1355.492} C_VEL
LIN {X 0,Y 587.363,Z 320.136,A -85,B 0,C 180,E1 -1358.254,E2 -1358.254} C_VEL
LIN {X 0,Y 587.35,Z 320.135,A -85,B 0,C 180,E1 -1361.141,E2 -1361.141} C_VEL
LIN {X 0,Y 587.352,Z 320.138,A -85,B 0,C 180,E1 -1364.26,E2 -1364.26} C_VEL
LIN {X 0,Y 587.349,Z 320.136,A -85,B 0,C 180,E1 -1367.405,E2 -1367.405} C_VEL
LIN {X 0,Y 587.326,Z 320.142,A -85,B 0,C 180,E1 -1370.304,E2 -1370.304} C_VEL
LIN {X 0,Y 587.313,Z 320.14,A -85,B 0,C 180,E1 -1373.258,E2 -1373.258} C_VEL
LIN {X 0,Y 587.324,Z 320.139,A -85,B 0,C 180,E1 -1375.516,E2 -1375.516} C_VEL
LIN {X 0,Y 587.337,Z 320.138,A -85,B 0,C 180,E1 -1377.817,E2 -1377.817} C_VEL
LIN {X 0,Y 587.34,Z 320.137,A -85,B 0,C 180,E1 -1380.513,E2 -1380.513} C_VEL
LIN {X 0,Y 587.328,Z 320.14,A -85,B 0,C 180,E1 -1383.396,E2 -1383.396} C_VEL
LIN {X 0,Y 587.345,Z 320.139,A -85,B 0,C 180,E1 -1385.895,E2 -1385.895} C_VEL
LIN {X 0,Y 587.319,Z 320.143,A -85,B 0,C 180,E1 -1388.479,E2 -1388.479} C_VEL
LIN {X 0,Y 587.348,Z 320.137,A -85,B 0,C 180,E1 -1391.154,E2 -1391.154} C_VEL
LIN {X 0,Y 587.319,Z 320.139,A -85,B 0,C 180,E1 -1394.114,E2 -1394.114} C_VEL
LIN {X 0,Y 587.308,Z 320.144,A -85,B 0,C 180,E1 -1396.995,E2 -1396.995} C_VEL
LIN {X 0,Y 587.316,Z 320.139,A -85,B 0,C 180,E1 -1399.98,E2 -1399.98} C_VEL
LIN {X 0,Y 587.336,Z 320.137,A -85,B 0,C 180,E1 -1402.393,E2 -1402.393} C_VEL
LIN {X 0,Y 587.338,Z 320.137,A -85,B 0,C 180,E1 -1404.946,E2 -1404.946} C_VEL
LIN {X 0,Y 587.327,Z 320.138,A -85,B 0,C 180,E1 -1407.421,E2 -1407.421} C_VEL
LIN {X 0,Y 587.335,Z 320.137,A -85,B 0,C 180,E1 -1409.831,E2 -1409.831} C_VEL
LIN {X 0,Y 587.338,Z 320.137,A -85,B 0,C 180,E1 -1412.307,E2 -1412.307} C_VEL
LIN {X 0,Y 587.338,Z 320.14,A -85,B 0,C 180,E1 -1415.242,E2 -1415.242} C_VEL
LIN {X 0,Y 587.357,Z 320.137,A -85,B 0,C 180,E1 -1417.488,E2 -1417.488} C_VEL
LIN {X 0,Y 587.333,Z 320.138,A -85,B 0,C 180,E1 -1420.426,E2 -1420.426} C_VEL
LIN {X 0,Y 587.345,Z 320.137,A -85,B 0,C 180,E1 -1423.312,E2 -1423.312} C_VEL
LIN {X 0,Y 587.348,Z 320.139,A -85,B 0,C 180,E1 -1426.155,E2 -1426.155} C_VEL
LIN {X 0,Y 587.331,Z 320.138,A -85,B 0,C 180,E1 -1428.963,E2 -1428.963} C_VEL
LIN {X 0,Y 587.366,Z 320.134,A -85,B 0,C 180,E1 -1431.746,E2 -1431.746} C_VEL
LIN {X 0,Y 587.354,Z 320.138,A -85,B 0,C 180,E1 -1434.508,E2 -1434.508} C_VEL
LIN {X 0,Y 587.374,Z 320.134,A -85,B 0,C 180,E1 -1437.257,E2 -1437.257} C_VEL
LIN {X 0,Y 587.368,Z 320.133,A -85,B 0,C 180,E1 -1440.001,E2 -1440.001} C_VEL
LIN {X 0,Y 587.362,Z 320.135,A -85,B 0,C 180,E1 -1442.744,E2 -1442.744} C_VEL
LIN {X 0,Y 587.351,Z 320.139,A -85,B 0,C 180,E1 -1445.494,E2 -1445.494} C_VEL
LIN {X 0,Y 587.358,Z 320.135,A -85,B 0,C 180,E1 -1448.256,E2 -1448.256} C_VEL
LIN {X 0,Y 587.352,Z 320.135,A -85,B 0,C 180,E1 -1451.142,E2 -1451.142} C_VEL
LIN {X 0,Y 587.356,Z 320.136,A -85,B 0,C 180,E1 -1454.262,E2 -1454.262} C_VEL
LIN {X 0,Y 587.352,Z 320.136,A -85,B 0,C 180,E1 -1457.406,E2 -1457.406} C_VEL
LIN {X 0,Y 587.324,Z 320.14,A -85,B 0,C 180,E1 -1460.305,E2 -1460.305} C_VEL
LIN {X 0,Y 587.317,Z 320.14,A -85,B 0,C 180,E1 -1463.259,E2 -1463.259} C_VEL
LIN {X 0,Y 587.326,Z 320.138,A -85,B 0,C 180,E1 -1465.517,E2 -1465.517} C_VEL
LIN {X 0,Y 587.341,Z 320.137,A -85,B 0,C 180,E1 -1467.818,E2 -1467.818} C_VEL
LIN {X 0,Y 587.337,Z 320.137,A -85,B 0,C 180,E1 -1470.512,E2 -1470.512} C_VEL
LIN {X 0,Y 587.33,Z 320.141,A -85,B 0,C 180,E1 -1473.397,E2 -1473.397} C_VEL
LIN {X 0,Y 587.351,Z 320.139,A -85,B 0,C 180,E1 -1475.896,E2 -1475.896} C_VEL
LIN {X 0,Y 587.328,Z 320.14,A -85,B 0,C 180,E1 -1478.48,E2 -1478.48} C_VEL
LIN {X 0,Y 587.329,Z 320.138,A -85,B 0,C 180,E1 -1481.158,E2 -1481.158} C_VEL
LIN {X 0,Y 587.328,Z 320.139,A -85,B 0,C 180,E1 -1484.115,E2 -1484.115} C_VEL
LIN {X 0,Y 587.314,Z 320.142,A -85,B 0,C 180,E1 -1486.995,E2 -1486.995} C_VEL
LIN {X 0,Y 587.312,Z 320.14,A -85,B 0,C 180,E1 -1489.747,E2 -1489.747} C_VEL
LIN {X 0,Y 587.342,Z 320.136,A -85,B 0,C 180,E1 -1492.394,E2 -1492.394} C_VEL
LIN {X 0,Y 587.349,Z 320.137,A -85,B 0,C 180,E1 -1494.947,E2 -1494.947} C_VEL
LIN {X 0,Y 587.386,Z 320.256,A -85,B 0,C 180,E1 -1496.83,E2 -1496.83} C_VEL
LIN {X 0,Y 587.602,Z 325.865,A -85,B 0,C 180,E1 -1498.65,E2 -1498.65} C_VEL
LIN {X 0,Y 587.453,Z 334.695,A -85,B 0,C 180,E1 -1501.411,E2 -1501.411} C_VEL
LIN {X 0,Y 587.45,Z 345.096,A -85,B 0,C 180,E1 -1504.49,E2 -1504.49} C_VEL
LIN {X 0,Y 587.352,Z 355.322,A -85,B 0,C 180,E1 -1507.488,E2 -1507.488} C_VEL
LIN {X 0,Y 587.32,Z 365.541,A -85,B 0,C 180,E1 -1510.425,E2 -1510.425} C_VEL
LIN {X 0,Y 587.282,Z 375.759,A -85,B 0,C 180,E1 -1513.31,E2 -1513.31} C_VEL
LIN {X 0,Y 587.223,Z 385.978,A -85,B 0,C 180,E1 -1516.152,E2 -1516.152} C_VEL
LIN {X 0,Y 587.201,Z 396.196,A -85,B 0,C 180,E1 -1518.961,E2 -1518.961} C_VEL
LIN {X 0,Y 587.196,Z 401.306,A -85,B 0,C 180,E1 -1520.355,E2 -1520.355} C_VEL
LIN {X 0,Y 587.498,Z 408.451,A -85,B 0,C 180,E1 -1520.534,E2 -1520.534} C_VEL
LIN {X 0,Y 587.463,Z 416.918,A -85,B 0,C 180,E1 -1520.794,E2 -1520.794} C_VEL
LIN {X 0,Y 587.402,Z 425.418,A -85,B 0,C 180,E1 -1521.14,E2 -1521.14} C_VEL
LIN {X 0,Y 587.378,Z 433.743,A -85,B 0,C 180,E1 -1521.573,E2 -1521.573} C_VEL
LIN {X 0,Y 587.327,Z 441.778,A -85,B 0,C 180,E1 -1522.091,E2 -1522.091} C_VEL
LIN {X 0,Y 587.291,Z 449.427,A -85,B 0,C 180,E1 -1522.696,E2 -1522.696} C_VEL
LIN {X 0,Y 587.281,Z 457.814,A -85,B 0,C 180,E1 -1523.513,E2 -1523.513} C_VEL
LIN {X 0,Y 587.238,Z 464.438,A -85,B 0,C 180,E1 -1524.335,E2 -1524.335} C_VEL
LIN {X 0,Y 587.17,Z 469.992,A -85,B 0,C 180,E1 -1525.195,E2 -1525.195} C_VEL
LIN {X 0,Y 587.21,Z 475.151,A -85,B 0,C 180,E1 -1526.227,E2 -1526.227} C_VEL
LIN {X 0,Y 587.155,Z 477.791,A -85,B 0,C 180,E1 -1526.913,E2 -1526.913} C_VEL
LIN {X 0,Y 587.141,Z 480.682,A -85,B 0,C 180,E1 -1527.943,E2 -1527.943} C_VEL
LIN {X 0,Y 587.145,Z 481.937,A -85,B 0,C 180,E1 -1528.629,E2 -1528.629} C_VEL
LIN {X 0,Y 587.136,Z 482.712,A -85,B 0,C 180,E1 -1529.315,E2 -1529.315} C_VEL
LIN {X 0,Y 587.134,Z 483,A -85,B 0,C 180,E1 -1530.001,E2 -1530.001} C_VEL
LIN {X 0,Y 587.136,Z 482.711,A -85,B 0,C 180,E1 -1530.687,E2 -1530.687} C_VEL
LIN {X 0,Y 587.145,Z 481.934,A -85,B 0,C 180,E1 -1531.373,E2 -1531.373} C_VEL
LIN {X 0,Y 587.141,Z 480.678,A -85,B 0,C 180,E1 -1532.059,E2 -1532.059} C_VEL
LIN {X 0,Y 587.155,Z 477.785,A -85,B 0,C 180,E1 -1533.088,E2 -1533.088} C_VEL
LIN {X 0,Y 587.21,Z 475.143,A -85,B 0,C 180,E1 -1533.775,E2 -1533.775} C_VEL
LIN {X 0,Y 587.17,Z 469.981,A -85,B 0,C 180,E1 -1534.807,E2 -1534.807} C_VEL
LIN {X 0,Y 587.253,Z 463.182,A -85,B 0,C 180,E1 -1535.839,E2 -1535.839} C_VEL
LIN {X 0,Y 587.27,Z 456.284,A -85,B 0,C 180,E1 -1536.646,E2 -1536.646} C_VEL
LIN {X 0,Y 587.292,Z 449.409,A -85,B 0,C 180,E1 -1537.306,E2 -1537.306} C_VEL
LIN {X 0,Y 587.332,Z 441.755,A -85,B 0,C 180,E1 -1537.91,E2 -1537.91} C_VEL
LIN {X 0,Y 587.379,Z 433.713,A -85,B 0,C 180,E1 -1538.429,E2 -1538.429} C_VEL
LIN {X 0,Y 587.403,Z 425.38,A -85,B 0,C 180,E1 -1538.862,E2 -1538.862} C_VEL
LIN {X 0,Y 587.44,Z 416.87,A -85,B 0,C 180,E1 -1539.209,E2 -1539.209} C_VEL
LIN {X 0,Y 587.49,Z 406.723,A -85,B 0,C 180,E1 -1539.512,E2 -1539.512} C_VEL
LIN {X 0,Y 587.197,Z 401.299,A -85,B 0,C 180,E1 -1539.647,E2 -1539.647} C_VEL
LIN {X 0,Y 587.229,Z 391.081,A -85,B 0,C 180,E1 -1542.441,E2 -1542.441} C_VEL
LIN {X 0,Y 587.246,Z 380.862,A -85,B 0,C 180,E1 -1545.266,E2 -1545.266} C_VEL
LIN {X 0,Y 587.303,Z 371.921,A -85,B 0,C 180,E1 -1547.768,E2 -1547.768} C_VEL
LIN {X 0,Y 587.332,Z 361.702,A -85,B 0,C 180,E1 -1550.671,E2 -1550.671} C_VEL
LIN {X 0,Y 587.383,Z 351.483,A -85,B 0,C 180,E1 -1553.631,E2 -1553.631} C_VEL
LIN {X 0,Y 587.437,Z 342.474,A -85,B 0,C 180,E1 -1556.275,E2 -1556.275} C_VEL
LIN {X 0,Y 587.458,Z 332.777,A -85,B 0,C 180,E1 -1559.152,E2 -1559.152} C_VEL
LIN {X 0,Y 587.596,Z 325.834,A -85,B 0,C 180,E1 -1561.352,E2 -1561.352} C_VEL
LIN {X 0,Y 587.394,Z 320.263,A -85,B 0,C 180,E1 -1563.173,E2 -1563.173} C_VEL
LIN {X 0,Y 587.295,Z 320.146,A -85,B 0,C 180,E1 -1565.9,E2 -1565.9} C_VEL
LIN {X 0,Y 587.326,Z 320.14,A -85,B 0,C 180,E1 -1568.48,E2 -1568.48} C_VEL
LIN {X 0,Y 587.34,Z 320.138,A -85,B 0,C 180,E1 -1571.157,E2 -1571.157} C_VEL
LIN {X 0,Y 587.326,Z 320.143,A -85,B 0,C 180,E1 -1574.113,E2 -1574.113} C_VEL
LIN {X 0,Y 587.32,Z 320.139,A -85,B 0,C 180,E1 -1576.994,E2 -1576.994} C_VEL
LIN {X 0,Y 587.317,Z 320.141,A -85,B 0,C 180,E1 -1579.746,E2 -1579.746} C_VEL
LIN {X 0,Y 587.346,Z 320.139,A -85,B 0,C 180,E1 -1582.392,E2 -1582.392} C_VEL
LIN {X 0,Y 587.348,Z 320.137,A -85,B 0,C 180,E1 -1585.653,E2 -1585.653} C_VEL
LIN {X 0,Y 587.342,Z 320.14,A -85,B 0,C 180,E1 -1588.231,E2 -1588.231} C_VEL
LIN {X 0,Y 587.354,Z 320.136,A -85,B 0,C 180,E1 -1590.867,E2 -1590.867} C_VEL
LIN {X 0,Y 587.345,Z 320.137,A -85,B 0,C 180,E1 -1593.823,E2 -1593.823} C_VEL
LIN {X 0,Y 587.327,Z 320.139,A -85,B 0,C 180,E1 -1595.993,E2 -1595.993} C_VEL
LIN {X 0,Y 587.322,Z 320.139,A -85,B 0,C 180,E1 -1598.225,E2 -1598.225} C_VEL
LIN {X 0,Y 587.35,Z 320.139,A -85,B 0,C 180,E1 -1601.151,E2 -1601.151} C_VEL
LIN {X 0,Y 587.323,Z 320.139,A -85,B 0,C 180,E1 -1604.024,E2 -1604.024} C_VEL
LIN {X 0,Y 587.32,Z 320.141,A -85,B 0,C 180,E1 -1606.858,E2 -1606.858} C_VEL
LIN {X 0,Y 587.339,Z 320.139,A -85,B 0,C 180,E1 -1609.66,E2 -1609.66} C_VEL
LIN {X 0,Y 587.369,Z 320.133,A -85,B 0,C 180,E1 -1612.436,E2 -1612.436} C_VEL
LIN {X 0,Y 587.367,Z 320.136,A -85,B 0,C 180,E1 -1615.195,E2 -1615.195} C_VEL
LIN {X 0,Y 587.365,Z 320.135,A -85,B 0,C 180,E1 -1617.942,E2 -1617.942} C_VEL
LIN {X 0,Y 587.396,Z 320.13,A -85,B 0,C 180,E1 -1620.685,E2 -1620.685} C_VEL
LIN {X 0,Y 587.327,Z 320.14,A -85,B 0,C 180,E1 -1623.429,E2 -1623.429} C_VEL
LIN {X 0,Y 587.352,Z 320.135,A -85,B 0,C 180,E1 -1625.492,E2 -1625.492} C_VEL
LIN {X 0,Y 587.359,Z 320.135,A -85,B 0,C 180,E1 -1627.562,E2 -1627.562} C_VEL
LIN {X 0,Y 587.345,Z 320.137,A -85,B 0,C 180,E1 -1630.339,E2 -1630.339} C_VEL
LIN {X 0,Y 587.317,Z 320.143,A -85,B 0,C 180,E1 -1633.141,E2 -1633.141} C_VEL
LIN {X 0,Y 587.326,Z 320.141,A -85,B 0,C 180,E1 -1635.321,E2 -1635.321} C_VEL
LIN {X 0,Y 587.307,Z 320.142,A -85,B 0,C 180,E1 -1637.406,E2 -1637.406} C_VEL
LIN {X 0,Y 587.228,Z 320.461,A -85,B 0,C 180,E1 -1638.308,E2 -1638.308} C_VEL
LIN {X 0,Y 586.566,Z 321.355,A -85,B 0,C 180,E1 -1638.873,E2 -1638.873} C_VEL
LIN {X 0,Y 583.703,Z 322.956,A -85,B 0,C 180,E1 -1639.789,E2 -1639.789} C_VEL
LIN {X 0,Y 581.284,Z 324.253,A -85,B 0,C 180,E1 -1640.525,E2 -1640.525} C_VEL
LIN {X 0,Y 580.252,Z 325.182,A -85,B 0,C 180,E1 -1641.094,E2 -1641.094} C_VEL
LIN {X 0,Y 580.171,Z 325.474,A -85,B 0,C 180,E1 -1641.287,E2 -1641.287} C_VEL
LIN {X 0,Y 580.146,Z 328.691,A -85,B 0,C 180,E1 -1643.563,E2 -1643.563} C_VEL
LIN {X 0,Y 580.124,Z 332.565,A -85,B 0,C 180,E1 -1646.299,E2 -1646.299} C_VEL
LIN {X 0,Y 580.073,Z 337.044,A -85,B 0,C 180,E1 -1649.268,E2 -1649.268} C_VEL
LIN {X 0,Y 580.042,Z 341.292,A -85,B 0,C 180,E1 -1651.989,E2 -1651.989} C_VEL
LIN {X 0,Y 580.027,Z 345.611,A -85,B 0,C 180,E1 -1654.713,E2 -1654.713} C_VEL
LIN {X 0,Y 580.013,Z 349.747,A -85,B 0,C 180,E1 -1657.289,E2 -1657.289} C_VEL
LIN {X 0,Y 580.043,Z 354.708,A -85,B 0,C 180,E1 -1660.345,E2 -1660.345} C_VEL
LIN {X 0,Y 580.489,Z 360.246,A -85,B 0,C 180,E1 -1660.511,E2 -1660.511} C_VEL
LIN {X 0,Y 580.437,Z 371.104,A -85,B 0,C 180,E1 -1660.88,E2 -1660.88} C_VEL
LIN {X 0,Y 580.363,Z 381.664,A -85,B 0,C 180,E1 -1661.393,E2 -1661.393} C_VEL
LIN {X 0,Y 580.279,Z 390.06,A -85,B 0,C 180,E1 -1661.916,E2 -1661.916} C_VEL
LIN {X 0,Y 580.25,Z 397.786,A -85,B 0,C 180,E1 -1662.51,E2 -1662.51} C_VEL
LIN {X 0,Y 580.219,Z 404.981,A -85,B 0,C 180,E1 -1663.184,E2 -1663.184} C_VEL
LIN {X 0,Y 580.169,Z 410.824,A -85,B 0,C 180,E1 -1663.843,E2 -1663.843} C_VEL
LIN {X 0,Y 580.152,Z 416.633,A -85,B 0,C 180,E1 -1664.636,E2 -1664.636} C_VEL
LIN {X 0,Y 580.134,Z 422.408,A -85,B 0,C 180,E1 -1665.621,E2 -1665.621} C_VEL
LIN {X 0,Y 580.08,Z 426.822,A -85,B 0,C 180,E1 -1666.628,E2 -1666.628} C_VEL
LIN {X 0,Y 580.071,Z 429.958,A -85,B 0,C 180,E1 -1667.65,E2 -1667.65} C_VEL
LIN {X 0,Y 580.031,Z 431.989,A -85,B 0,C 180,E1 -1668.695,E2 -1668.695} C_VEL
LIN {X 0,Y 580.013,Z 432.568,A -85,B 0,C 180,E1 -1669.131,E2 -1669.131} C_VEL
LIN {X 0,Y 580.036,Z 433,A -85,B 0,C 180,E1 -1670.045,E2 -1670.045} C_VEL
LIN {X 0,Y 580.005,Z 432.584,A -85,B 0,C 180,E1 -1670.942,E2 -1670.942} C_VEL
LIN {X 0,Y 580.036,Z 431.074,A -85,B 0,C 180,E1 -1671.957,E2 -1671.957} C_VEL
LIN {X 0,Y 580.053,Z 429.284,A -85,B 0,C 180,E1 -1672.712,E2 -1672.712} C_VEL
LIN {X 0,Y 580.081,Z 426.374,A -85,B 0,C 180,E1 -1673.582,E2 -1673.582} C_VEL
LIN {X 0,Y 580.108,Z 421.388,A -85,B 0,C 180,E1 -1674.655,E2 -1674.655} C_VEL
LIN {X 0,Y 580.133,Z 416.577,A -85,B 0,C 180,E1 -1675.463,E2 -1675.463} C_VEL
LIN {X 0,Y 580.143,Z 410.496,A -85,B 0,C 180,E1 -1676.287,E2 -1676.287} C_VEL
LIN {X 0,Y 580.224,Z 404.354,A -85,B 0,C 180,E1 -1676.97,E2 -1676.97} C_VEL
LIN {X 0,Y 580.257,Z 396.454,A -85,B 0,C 180,E1 -1677.694,E2 -1677.694} C_VEL
LIN {X 0,Y 580.305,Z 386.521,A -85,B 0,C 180,E1 -1678.412,E2 -1678.412} C_VEL
LIN {X 0,Y 580.369,Z 378.019,A -85,B 0,C 180,E1 -1678.891,E2 -1678.891} C_VEL
LIN {X 0,Y 580.438,Z 369.282,A -85,B 0,C 180,E1 -1679.278,E2 -1679.278} C_VEL
LIN {X 0,Y 580.489,Z 359.494,A -85,B 0,C 180,E1 -1679.599,E2 -1679.599} C_VEL
LIN {X 0,Y 580.067,Z 354.718,A -85,B 0,C 180,E1 -1679.738,E2 -1679.738} C_VEL
LIN {X 0,Y 580.058,Z 350.094,A -85,B 0,C 180,E1 -1682.586,E2 -1682.586} C_VEL
LIN {X 0,Y 580.079,Z 345.702,A -85,B 0,C 180,E1 -1685.319,E2 -1685.319} C_VEL
LIN {X 0,Y 580.04,Z 341.55,A -85,B 0,C 180,E1 -1687.937,E2 -1687.937} C_VEL
LIN {X 0,Y 580.064,Z 338.057,A -85,B 0,C 180,E1 -1690.168,E2 -1690.168} C_VEL
LIN {X 0,Y 580.119,Z 333.504,A -85,B 0,C 180,E1 -1693.145,E2 -1693.145} C_VEL
LIN {X 0,Y 580.103,Z 329.501,A -85,B 0,C 180,E1 -1695.977,E2 -1695.977} C_VEL
LIN {X 0,Y 580.202,Z 325.242,A -85,B 0,C 180,E1 -1698.852,E2 -1698.852} C_VEL
LIN {X 0,Y 580.185,Z 321.228,A -85,B 0,C 180,E1 -1701.641,E2 -1701.641} C_VEL
LIN {X 0,Y 580.269,Z 321.019,A -85,B 0,C 180,E1 -1703.741,E2 -1703.741} C_VEL
LIN {X 0,Y 580.269,Z 321.02,A -85,B 0,C 180,E1 -1705.832,E2 -1705.832} C_VEL
LIN {X 0,Y 580.324,Z 321.011,A -85,B 0,C 180,E1 -1707.917,E2 -1707.917} C_VEL
LIN {X 0,Y 580.357,Z 321.009,A -85,B 0,C 180,E1 -1710.693,E2 -1710.693} C_VEL
LIN {X 0,Y 580.282,Z 321.018,A -85,B 0,C 180,E1 -1713.471,E2 -1713.471} C_VEL
LIN {X 0,Y 580.319,Z 321.013,A -85,B 0,C 180,E1 -1715.559,E2 -1715.559} C_VEL
LIN {X 0,Y 580.327,Z 321.011,A -85,B 0,C 180,E1 -1718.355,E2 -1718.355} C_VEL
LIN {X 0,Y 580.321,Z 321.011,A -85,B 0,C 180,E1 -1721.208,E2 -1721.208} C_VEL
LIN {X 0,Y 580.303,Z 321.015,A -85,B 0,C 180,E1 -1724.338,E2 -1724.338} C_VEL
LIN {X 0,Y 580.301,Z 321.015,A -85,B 0,C 180,E1 -1726.914,E2 -1726.914} C_VEL
LIN {X 0,Y 580.297,Z 321.014,A -85,B 0,C 180,E1 -1729.821,E2 -1729.821} C_VEL
LIN {X 0,Y 580.264,Z 321.018,A -85,B 0,C 180,E1 -1732.052,E2 -1732.052} C_VEL
LIN {X 0,Y 580.295,Z 321.017,A -85,B 0,C 180,E1 -1735.079,E2 -1735.079} C_VEL
LIN {X 0,Y 580.307,Z 321.013,A -85,B 0,C 180,E1 -1737.863,E2 -1737.863} C_VEL
LIN {X 0,Y 580.288,Z 321.015,A -85,B 0,C 180,E1 -1740.697,E2 -1740.697} C_VEL
LIN {X 0,Y 580.295,Z 321.015,A -85,B 0,C 180,E1 -1743.317,E2 -1743.317} C_VEL
LIN {X 0,Y 580.314,Z 321.013,A -85,B 0,C 180,E1 -1745.768,E2 -1745.768} C_VEL
LIN {X 0,Y 580.275,Z 321.017,A -85,B 0,C 180,E1 -1748.146,E2 -1748.146} C_VEL
LIN {X 0,Y 580.306,Z 321.016,A -85,B 0,C 180,E1 -1750.841,E2 -1750.841} C_VEL
LIN {X 0,Y 580.276,Z 321.017,A -85,B 0,C 180,E1 -1753.656,E2 -1753.656} C_VEL
LIN {X 0,Y 580.271,Z 321.018,A -85,B 0,C 180,E1 -1756.608,E2 -1756.608} C_VEL
LIN {X 0,Y 580.29,Z 321.017,A -85,B 0,C 180,E1 -1759.157,E2 -1759.157} C_VEL
LIN {X 0,Y 580.28,Z 321.019,A -85,B 0,C 180,E1 -1761.926,E2 -1761.926} C_VEL
LIN {X 0,Y 580.294,Z 321.016,A -85,B 0,C 180,E1 -1764.457,E2 -1764.457} C_VEL
LIN {X 0,Y 580.279,Z 321.017,A -85,B 0,C 180,E1 -1766.976,E2 -1766.976} C_VEL
LIN {X 0,Y 580.298,Z 321.014,A -85,B 0,C 180,E1 -1769.426,E2 -1769.426} C_VEL
LIN {X 0,Y 580.307,Z 321.013,A -85,B 0,C 180,E1 -1772.137,E2 -1772.137} C_VEL
LIN {X 0,Y 580.308,Z 321.015,A -85,B 0,C 180,E1 -1775.27,E2 -1775.27} C_VEL
LIN {X 0,Y 580.278,Z 321.017,A -85,B 0,C 180,E1 -1777.949,E2 -1777.949} C_VEL
LIN {X 0,Y 580.305,Z 321.014,A -85,B 0,C 180,E1 -1780.915,E2 -1780.915} C_VEL
LIN {X 0,Y 580.273,Z 321.019,A -85,B 0,C 180,E1 -1783.826,E2 -1783.826} C_VEL
LIN {X 0,Y 580.314,Z 321.014,A -85,B 0,C 180,E1 -1785.984,E2 -1785.984} C_VEL
LIN {X 0,Y 580.291,Z 321.015,A -85,B 0,C 180,E1 -1788.827,E2 -1788.827} C_VEL
LIN {X 0,Y 580.328,Z 321.01,A -85,B 0,C 180,E1 -1791.645,E2 -1791.645} C_VEL
LIN {X 0,Y 580.319,Z 321.014,A -85,B 0,C 180,E1 -1794.441,E2 -1794.441} C_VEL
LIN {X 0,Y 580.339,Z 321.011,A -85,B 0,C 180,E1 -1797.224,E2 -1797.224} C_VEL
LIN {X 0,Y 580.338,Z 321.009,A -85,B 0,C 180,E1 -1800.001,E2 -1800.001} C_VEL
LIN {X 0,Y 580.329,Z 321.011,A -85,B 0,C 180,E1 -1802.777,E2 -1802.777} C_VEL
LIN {X 0,Y 580.317,Z 321.015,A -85,B 0,C 180,E1 -1805.56,E2 -1805.56} C_VEL
LIN {X 0,Y 580.321,Z 321.011,A -85,B 0,C 180,E1 -1808.357,E2 -1808.357} C_VEL
LIN {X 0,Y 580.323,Z 321.011,A -85,B 0,C 180,E1 -1811.209,E2 -1811.209} C_VEL
LIN {X 0,Y 580.306,Z 321.013,A -85,B 0,C 180,E1 -1814.34,E2 -1814.34} C_VEL
LIN {X 0,Y 580.306,Z 321.013,A -85,B 0,C 180,E1 -1816.916,E2 -1816.916} C_VEL
LIN {X 0,Y 580.299,Z 321.015,A -85,B 0,C 180,E1 -1819.823,E2 -1819.823} C_VEL
LIN {X 0,Y 580.29,Z 321.016,A -85,B 0,C 180,E1 -1822.803,E2 -1822.803} C_VEL
LIN {X 0,Y 580.298,Z 321.016,A -85,B 0,C 180,E1 -1825.081,E2 -1825.081} C_VEL
LIN {X 0,Y 580.312,Z 321.012,A -85,B 0,C 180,E1 -1827.864,E2 -1827.864} C_VEL
LIN {X 0,Y 580.283,Z 321.016,A -85,B 0,C 180,E1 -1830.697,E2 -1830.697} C_VEL
LIN {X 0,Y 580.299,Z 321.016,A -85,B 0,C 180,E1 -1833.318,E2 -1833.318} C_VEL
LIN {X 0,Y 580.321,Z 321.014,A -85,B 0,C 180,E1 -1835.769,E2 -1835.769} C_VEL
LIN {X 0,Y 580.283,Z 321.018,A -85,B 0,C 180,E1 -1838.147,E2 -1838.147} C_VEL
LIN {X 0,Y 580.292,Z 321.017,A -85,B 0,C 180,E1 -1840.844,E2 -1840.844} C_VEL
LIN {X 0,Y 580.282,Z 321.016,A -85,B 0,C 180,E1 -1843.658,E2 -1843.658} C_VEL
LIN {X 0,Y 580.279,Z 321.018,A -85,B 0,C 180,E1 -1846.609,E2 -1846.609} C_VEL
LIN {X 0,Y 580.296,Z 321.017,A -85,B 0,C 180,E1 -1849.158,E2 -1849.158} C_VEL
LIN {X 0,Y 580.286,Z 321.016,A -85,B 0,C 180,E1 -1851.928,E2 -1851.928} C_VEL
LIN {X 0,Y 580.305,Z 321.014,A -85,B 0,C 180,E1 -1854.458,E2 -1854.458} C_VEL
LIN {X 0,Y 580.336,Z 321.169,A -85,B 0,C 180,E1 -1856.679,E2 -1856.679} C_VEL
LIN {X 0,Y 580.613,Z 324.903,A -85,B 0,C 180,E1 -1857.921,E2 -1857.921} C_VEL
LIN {X 0,Y 580.49,Z 333.382,A -85,B 0,C 180,E1 -1860.658,E2 -1860.658} C_VEL
LIN {X 0,Y 580.391,Z 342.398,A -85,B 0,C 180,E1 -1863.384,E2 -1863.384} C_VEL
LIN {X 0,Y 580.355,Z 351.486,A -85,B 0,C 180,E1 -1866.068,E2 -1866.068} C_VEL
LIN {X 0,Y 580.301,Z 360.906,A -85,B 0,C 180,E1 -1868.835,E2 -1868.835} C_VEL
LIN {X 0,Y 580.235,Z 370.65,A -85,B 0,C 180,E1 -1871.645,E2 -1871.645} C_VEL
LIN {X 0,Y 580.187,Z 379.591,A -85,B 0,C 180,E1 -1874.185,E2 -1874.185} C_VEL
LIN {X 0,Y 580.163,Z 388.533,A -85,B 0,C 180,E1 -1876.694,E2 -1876.694} C_VEL
LIN {X 0,Y 580.152,Z 397.575,A -85,B 0,C 180,E1 -1879.206,E2 -1879.206} C_VEL
LIN {X 0,Y 580.116,Z 401.306,A -85,B 0,C 180,E1 -1880.236,E2 -1880.236} C_VEL
LIN {X 0,Y 580.509,Z 408.451,A -85,B 0,C 180,E1 -1880.419,E2 -1880.419} C_VEL
LIN {X 0,Y 580.465,Z 416.92,A -85,B 0,C 180,E1 -1880.682,E2 -1880.682} C_VEL
LIN {X 0,Y 580.406,Z 425.421,A -85,B 0,C 180,E1 -1881.032,E2 -1881.032} C_VEL
LIN {X 0,Y 580.359,Z 433.746,A -85,B 0,C 180,E1 -1881.47,E2 -1881.47} C_VEL
LIN {X 0,Y 580.278,Z 441.78,A -85,B 0,C 180,E1 -1881.995,E2 -1881.995} C_VEL
LIN {X 0,Y 580.239,Z 449.428,A -85,B 0,C 180,E1 -1882.607,E2 -1882.607} C_VEL
LIN {X 0,Y 580.216,Z 456.892,A -85,B 0,C 180,E1 -1883.336,E2 -1883.336} C_VEL
LIN {X 0,Y 580.173,Z 464.439,A -85,B 0,C 180,E1 -1884.265,E2 -1884.265} C_VEL
LIN {X 0,Y 580.084,Z 469.992,A -85,B 0,C 180,E1 -1885.136,E2 -1885.136} C_VEL
LIN {X 0,Y 580.136,Z 475.152,A -85,B 0,C 180,E1 -1886.181,E2 -1886.181} C_VEL
LIN {X 0,Y 580.07,Z 477.792,A -85,B 0,C 180,E1 -1886.876,E2 -1886.876} C_VEL
LIN {X 0,Y 580.041,Z 480.683,A -85,B 0,C 180,E1 -1887.918,E2 -1887.918} C_VEL
LIN {X 0,Y 580.045,Z 481.938,A -85,B 0,C 180,E1 -1888.612,E2 -1888.612} C_VEL
LIN {X 0,Y 580.036,Z 482.712,A -85,B 0,C 180,E1 -1889.307,E2 -1889.307} C_VEL
LIN {X 0,Y 580.034,Z 483,A -85,B 0,C 180,E1 -1890.001,E2 -1890.001} C_VEL
LIN {X 0,Y 580.036,Z 482.711,A -85,B 0,C 180,E1 -1890.695,E2 -1890.695} C_VEL
LIN {X 0,Y 580.045,Z 481.935,A -85,B 0,C 180,E1 -1891.389,E2 -1891.389} C_VEL
LIN {X 0,Y 580.041,Z 480.678,A -85,B 0,C 180,E1 -1892.084,E2 -1892.084} C_VEL
LIN {X 0,Y 580.07,Z 477.785,A -85,B 0,C 180,E1 -1893.126,E2 -1893.126} C_VEL
LIN {X 0,Y 580.122,Z 475.144,A -85,B 0,C 180,E1 -1893.821,E2 -1893.821} C_VEL
LIN {X 0,Y 580.084,Z 469.981,A -85,B 0,C 180,E1 -1894.866,E2 -1894.866} C_VEL
LIN {X 0,Y 580.193,Z 463.181,A -85,B 0,C 180,E1 -1895.911,E2 -1895.911} C_VEL
LIN {X 0,Y 580.226,Z 455.492,A -85,B 0,C 180,E1 -1896.808,E2 -1896.808} C_VEL
LIN {X 0,Y 580.254,Z 448.396,A -85,B 0,C 180,E1 -1897.482,E2 -1897.482} C_VEL
LIN {X 0,Y 580.296,Z 440.536,A -85,B 0,C 180,E1 -1898.094,E2 -1898.094} C_VEL
LIN {X 0,Y 580.39,Z 430.719,A -85,B 0,C 180,E1 -1898.707,E2 -1898.707} C_VEL
LIN {X 0,Y 580.451,Z 419.278,A -85,B 0,C 180,E1 -1899.233,E2 -1899.233} C_VEL
LIN {X 0,Y 580.512,Z 409.215,A -85,B 0,C 180,E1 -1899.561,E2 -1899.561} C_VEL
LIN {X 0,Y 580.222,Z 402.341,A -85,B 0,C 180,E1 -1899.731,E2 -1899.731} C_VEL
LIN {X 0,Y 580.117,Z 401.299,A -85,B 0,C 180,E1 -1899.766,E2 -1899.766} C_VEL
LIN {X 0,Y 580.17,Z 391.081,A -85,B 0,C 180,E1 -1902.595,E2 -1902.595} C_VEL
LIN {X 0,Y 580.183,Z 380.862,A -85,B 0,C 180,E1 -1905.457,E2 -1905.457} C_VEL
LIN {X 0,Y 580.254,Z 371.921,A -85,B 0,C 180,E1 -1907.991,E2 -1907.991} C_VEL
LIN {X 0,Y 580.287,Z 361.94,A -85,B 0,C 180,E1 -1910.865,E2 -1910.865} C_VEL
LIN {X 0,Y 580.366,Z 352.761,A -85,B 0,C 180,E1 -1913.555,E2 -1913.555} C_VEL
LIN {X 0,Y 580.404,Z 343.222,A -85,B 0,C 180,E1 -1916.356,E2 -1916.356} C_VEL
LIN {X 0,Y 580.434,Z 334.547,A -85,B 0,C 180,E1 -1918.969,E2 -1918.969} C_VEL
LIN {X 0,Y 580.605,Z 327.062,A -85,B 0,C 180,E1 -1921.366,E2 -1921.366} C_VEL
LIN {X 0,Y 580.496,Z 322.068,A -85,B 0,C 180,E1 -1923.012,E2 -1923.012} C_VEL
LIN {X 0,Y 580.328,Z 321.014,A -85,B 0,C 180,E1 -1923.404,E2 -1923.404} C_VEL
LIN {X 0,Y 580.272,Z 321.018,A -85,B 0,C 180,E1 -1926.404,E2 -1926.404} C_VEL
LIN {X 0,Y 580.293,Z 321.017,A -85,B 0,C 180,E1 -1929.185,E2 -1929.185} C_VEL
LIN {X 0,Y 580.283,Z 321.02,A -85,B 0,C 180,E1 -1931.769,E2 -1931.769} C_VEL
LIN {X 0,Y 580.256,Z 321.02,A -85,B 0,C 180,E1 -1934.628,E2 -1934.628} C_VEL
LIN {X 0,Y 580.292,Z 321.018,A -85,B 0,C 180,E1 -1937.628,E2 -1937.628} C_VEL
LIN {X 0,Y 580.287,Z 321.018,A -85,B 0,C 180,E1 -1940.066,E2 -1940.066} C_VEL
LIN {X 0,Y 580.303,Z 321.014,A -85,B 0,C 180,E1 -1943.066,E2 -1943.066} C_VEL
LIN {X 0,Y 580.305,Z 321.014,A -85,B 0,C 180,E1 -1946.144,E2 -1946.144} C_VEL
LIN {X 0,Y 580.276,Z 321.017,A -85,B 0,C 180,E1 -1948.614,E2 -1948.614} C_VEL
LIN {X 0,Y 580.297,Z 321.014,A -85,B 0,C 180,E1 -1951.024,E2 -1951.024} C_VEL
LIN {X 0,Y 580.296,Z 321.015,A -85,B 0,C 180,E1 -1953.666,E2 -1953.666} C_VEL
LIN {X 0,Y 580.3,Z 321.014,A -85,B 0,C 180,E1 -1955.683,E2 -1955.683} C_VEL
LIN {X 0,Y 580.275,Z 321.018,A -85,B 0,C 180,E1 -1957.947,E2 -1957.947} C_VEL
LIN {X 0,Y 580.303,Z 321.015,A -85,B 0,C 180,E1 -1960.913,E2 -1960.913} C_VEL
LIN {X 0,Y 580.279,Z 321.017,A -85,B 0,C 180,E1 -1963.825,E2 -1963.825} C_VEL
LIN {X 0,Y 580.278,Z 321.017,A -85,B 0,C 180,E1 -1966.695,E2 -1966.695} C_VEL
LIN {X 0,Y 580.311,Z 321.012,A -85,B 0,C 180,E1 -1968.826,E2 -1968.826} C_VEL
LIN {X 0,Y 580.314,Z 321.014,A -85,B 0,C 180,E1 -1971.643,E2 -1971.643} C_VEL
LIN {X 0,Y 580.327,Z 321.012,A -85,B 0,C 180,E1 -1974.44,E2 -1974.44} C_VEL
LIN {X 0,Y 580.334,Z 321.01,A -85,B 0,C 180,E1 -1977.223,E2 -1977.223} C_VEL
LIN {X 0,Y 580.355,Z 321.01,A -85,B 0,C 180,E1 -1979.999,E2 -1979.999} C_VEL
LIN {X 0,Y 580.341,Z 321.009,A -85,B 0,C 180,E1 -1982.776,E2 -1982.776} C_VEL
LIN {X 0,Y 580.32,Z 321.012,A -85,B 0,C 180,E1 -1985.559,E2 -1985.559} C_VEL
LIN {X 0,Y 580.32,Z 321.011,A -85,B 0,C 180,E1 -1987.655,E2 -1987.655} C_VEL
LIN {X 0,Y 580.304,Z 321.015,A -85,B 0,C 180,E1 -1990.466,E2 -1990.466} C_VEL
LIN {X 0,Y 580.274,Z 321.019,A -85,B 0,C 180,E1 -1993.303,E2 -1993.303} C_VEL
LIN {X 0,Y 580.296,Z 321.018,A -85,B 0,C 180,E1 -1995.452,E2 -1995.452} C_VEL
LIN {X 0,Y 580.247,Z 321.023,A -85,B 0,C 180,E1 -1997.625,E2 -1997.625} C_VEL
LIN {X 0,Y 580.162,Z 321.215,A -85,B 0,C 180,E1 -1998.357,E2 -1998.357} C_VEL
LIN {X 0,Y 580.171,Z 325.474,A -85,B 0,C 180,E1 -2001.287,E2 -2001.287} C_VEL
LIN {X 0,Y 579.504,Z 326.387,A -85,B 0,C 180,E1 -2001.86,E2 -2001.86} C_VEL
LIN {X 0,Y 576.611,Z 327.946,A -85,B 0,C 180,E1 -2002.787,E2 -2002.787} C_VEL
LIN {X 0,Y 574.167,Z 329.196,A -85,B 0,C 180,E1 -2003.534,E2 -2003.534} C_VEL
LIN {X 0,Y 573.127,Z 330.083,A -85,B 0,C 180,E1 -2004.111,E2 -2004.111} C_VEL
LIN {X 0,Y 573.047,Z 330.361,A -85,B 0,C 180,E1 -2004.307,E2 -2004.307} C_VEL
LIN {X 0,Y 573.002,Z 334.141,A -85,B 0,C 180,E1 -2006.987,E2 -2006.987} C_VEL
LIN {X 0,Y 572.976,Z 337.716,A -85,B 0,C 180,E1 -2009.439,E2 -2009.439} C_VEL
LIN {X 0,Y 572.953,Z 341.948,A -85,B 0,C 180,E1 -2012.18,E2 -2012.18} C_VEL
LIN {X 0,Y 572.948,Z 345.942,A -85,B 0,C 180,E1 -2014.729,E2 -2014.729} C_VEL
LIN {X 0,Y 572.906,Z 350.871,A -85,B 0,C 180,E1 -2017.832,E2 -2017.832} C_VEL
LIN {X 0,Y 572.951,Z 354.72,A -85,B 0,C 180,E1 -2020.232,E2 -2020.232} C_VEL
LIN {X 0,Y 573.5,Z 361.842,A -85,B 0,C 180,E1 -2020.436,E2 -2020.436} C_VEL
LIN {X 0,Y 573.404,Z 373.376,A -85,B 0,C 180,E1 -2020.869,E2 -2020.869} C_VEL
LIN {X 0,Y 573.337,Z 382.189,A -85,B 0,C 180,E1 -2021.317,E2 -2021.317} C_VEL
LIN {X 0,Y 573.241,Z 390.789,A -85,B 0,C 180,E1 -2021.869,E2 -2021.869} C_VEL
LIN {X 0,Y 573.189,Z 397.63,A -85,B 0,C 180,E1 -2022.404,E2 -2022.404} C_VEL
LIN {X 0,Y 573.184,Z 403.749,A -85,B 0,C 180,E1 -2022.972,E2 -2022.972} C_VEL
LIN {X 0,Y 573.106,Z 409.918,A -85,B 0,C 180,E1 -2023.654,E2 -2023.654} C_VEL
LIN {X 0,Y 573.067,Z 416.189,A -85,B 0,C 180,E1 -2024.502,E2 -2024.502} C_VEL
LIN {X 0,Y 573.058,Z 421.18,A -85,B 0,C 180,E1 -2025.34,E2 -2025.34} C_VEL
LIN {X 0,Y 572.983,Z 425.922,A -85,B 0,C 180,E1 -2026.357,E2 -2026.357} C_VEL
LIN {X 0,Y 572.995,Z 429.857,A -85,B 0,C 180,E1 -2027.576,E2 -2027.576} C_VEL
LIN {X 0,Y 572.943,Z 431.767,A -85,B 0,C 180,E1 -2028.517,E2 -2028.517} C_VEL
LIN {X 0,Y 572.935,Z 432.786,A -85,B 0,C 180,E1 -2029.509,E2 -2029.509} C_VEL
LIN {X 0,Y 572.913,Z 432.774,A -85,B 0,C 180,E1 -2030.607,E2 -2030.607} C_VEL
LIN {X 0,Y 572.937,Z 431.56,A -85,B 0,C 180,E1 -2031.725,E2 -2031.725} C_VEL
LIN {X 0,Y 572.997,Z 428.282,A -85,B 0,C 180,E1 -2033.058,E2 -2033.058} C_VEL
LIN {X 0,Y 573.001,Z 424.578,A -85,B 0,C 180,E1 -2034.046,E2 -2034.046} C_VEL
LIN {X 0,Y 573.004,Z 420.928,A -85,B 0,C 180,E1 -2034.797,E2 -2034.797} C_VEL
LIN {X 0,Y 573.056,Z 417.086,A -85,B 0,C 180,E1 -2035.454,E2 -2035.454} C_VEL
LIN {X 0,Y 573.08,Z 411.064,A -85,B 0,C 180,E1 -2036.294,E2 -2036.294} C_VEL
LIN {X 0,Y 573.176,Z 404.544,A -85,B 0,C 180,E1 -2037.036,E2 -2037.036} C_VEL
LIN {X 0,Y 573.21,Z 397.302,A -85,B 0,C 180,E1 -2037.714,E2 -2037.714} C_VEL
LIN {X 0,Y 573.269,Z 388.416,A -85,B 0,C 180,E1 -2038.392,E2 -2038.392} C_VEL
LIN {X 0,Y 573.342,Z 377.752,A -85,B 0,C 180,E1 -2039.013,E2 -2039.013} C_VEL
LIN {X 0,Y 573.428,Z 368.33,A -85,B 0,C 180,E1 -2039.427,E2 -2039.427} C_VEL
LIN {X 0,Y 573.466,Z 358.857,A -85,B 0,C 180,E1 -2039.734,E2 -2039.734} C_VEL
LIN {X 0,Y 572.978,Z 354.72,A -85,B 0,C 180,E1 -2039.858,E2 -2039.858} C_VEL
LIN {X 0,Y 572.958,Z 349.672,A -85,B 0,C 180,E1 -2043.008,E2 -2043.008} C_VEL
LIN {X 0,Y 572.996,Z 345.954,A -85,B 0,C 180,E1 -2045.353,E2 -2045.353} C_VEL
LIN {X 0,Y 572.953,Z 342.354,A -85,B 0,C 180,E1 -2047.65,E2 -2047.65} C_VEL
LIN {X 0,Y 573.008,Z 337.7,A -85,B 0,C 180,E1 -2050.66,E2 -2050.66} C_VEL
LIN {X 0,Y 573.032,Z 333.468,A -85,B 0,C 180,E1 -2053.614,E2 -2053.614} C_VEL
LIN {X 0,Y 573.019,Z 329.258,A -85,B 0,C 180,E1 -2056.524,E2 -2056.524} C_VEL
LIN {X 0,Y 573.12,Z 325.071,A -85,B 0,C 180,E1 -2059.4,E2 -2059.4} C_VEL
LIN {X 0,Y 573.124,Z 322.04,A -85,B 0,C 180,E1 -2061.537,E2 -2061.537} C_VEL
LIN {X 0,Y 573.232,Z 321.897,A -85,B 0,C 180,E1 -2063.664,E2 -2063.664} C_VEL
LIN {X 0,Y 573.226,Z 321.896,A -85,B 0,C 180,E1 -2065.78,E2 -2065.78} C_VEL
LIN {X 0,Y 573.296,Z 321.886,A -85,B 0,C 180,E1 -2067.891,E2 -2067.891} C_VEL
LIN {X 0,Y 573.327,Z 321.885,A -85,B 0,C 180,E1 -2070.701,E2 -2070.701} C_VEL
LIN {X 0,Y 573.234,Z 321.895,A -85,B 0,C 180,E1 -2073.514,E2 -2073.514} C_VEL
LIN {X 0,Y 573.286,Z 321.89,A -85,B 0,C 180,E1 -2075.627,E2 -2075.627} C_VEL
LIN {X 0,Y 573.298,Z 321.886,A -85,B 0,C 180,E1 -2078.458,E2 -2078.458} C_VEL
LIN {X 0,Y 573.287,Z 321.887,A -85,B 0,C 180,E1 -2081.311,E2 -2081.311} C_VEL
LIN {X 0,Y 573.269,Z 321.89,A -85,B 0,C 180,E1 -2084.424,E2 -2084.424} C_VEL
LIN {X 0,Y 573.247,Z 321.892,A -85,B 0,C 180,E1 -2087.111,E2 -2087.111} C_VEL
LIN {X 0,Y 573.248,Z 321.894,A -85,B 0,C 180,E1 -2090.076,E2 -2090.076} C_VEL
LIN {X 0,Y 573.227,Z 321.895,A -85,B 0,C 180,E1 -2092.337,E2 -2092.337} C_VEL
LIN {X 0,Y 573.242,Z 321.894,A -85,B 0,C 180,E1 -2095.409,E2 -2095.409} C_VEL
LIN {X 0,Y 573.253,Z 321.891,A -85,B 0,C 180,E1 -2098.032,E2 -2098.032} C_VEL
LIN {X 0,Y 573.233,Z 321.895,A -85,B 0,C 180,E1 -2100.885,E2 -2100.885} C_VEL
LIN {X 0,Y 573.273,Z 321.892,A -85,B 0,C 180,E1 -2103.528,E2 -2103.528} C_VEL
LIN {X 0,Y 573.248,Z 321.895,A -85,B 0,C 180,E1 -2106.048,E2 -2106.048} C_VEL
LIN {X 0,Y 573.235,Z 321.895,A -85,B 0,C 180,E1 -2108.701,E2 -2108.701} C_VEL
LIN {X 0,Y 573.25,Z 321.892,A -85,B 0,C 180,E1 -2111.597,E2 -2111.597} C_VEL
LIN {X 0,Y 573.224,Z 321.896,A -85,B 0,C 180,E1 -2114.333,E2 -2114.333} C_VEL
LIN {X 0,Y 573.228,Z 321.895,A -85,B 0,C 180,E1 -2117.358,E2 -2117.358} C_VEL
LIN {X 0,Y 573.238,Z 321.895,A -85,B 0,C 180,E1 -2120.394,E2 -2120.394} C_VEL
LIN {X 0,Y 573.244,Z 321.896,A -85,B 0,C 180,E1 -2123.078,E2 -2123.078} C_VEL
LIN {X 0,Y 573.263,Z 321.892,A -85,B 0,C 180,E1 -2125.672,E2 -2125.672} C_VEL
LIN {X 0,Y 573.236,Z 321.895,A -85,B 0,C 180,E1 -2128.186,E2 -2128.186} C_VEL
LIN {X 0,Y 573.259,Z 321.892,A -85,B 0,C 180,E1 -2130.635,E2 -2130.635} C_VEL
LIN {X 0,Y 573.24,Z 321.894,A -85,B 0,C 180,E1 -2133.025,E2 -2133.025} C_VEL
LIN {X 0,Y 573.262,Z 321.892,A -85,B 0,C 180,E1 -2135.367,E2 -2135.367} C_VEL
LIN {X 0,Y 573.247,Z 321.895,A -85,B 0,C 180,E1 -2137.664,E2 -2137.664} C_VEL
LIN {X 0,Y 573.266,Z 321.89,A -85,B 0,C 180,E1 -2140.728,E2 -2140.728} C_VEL
LIN {X 0,Y 573.248,Z 321.895,A -85,B 0,C 180,E1 -2143.623,E2 -2143.623} C_VEL
LIN {X 0,Y 573.226,Z 321.895,A -85,B 0,C 180,E1 -2146.53,E2 -2146.53} C_VEL
LIN {X 0,Y 573.249,Z 321.893,A -85,B 0,C 180,E1 -2148.746,E2 -2148.746} C_VEL
LIN {X 0,Y 573.299,Z 321.886,A -85,B 0,C 180,E1 -2151.542,E2 -2151.542} C_VEL
LIN {X 0,Y 573.286,Z 321.889,A -85,B 0,C 180,E1 -2154.373,E2 -2154.373} C_VEL
LIN {X 0,Y 573.307,Z 321.885,A -85,B 0,C 180,E1 -2157.893,E2 -2157.893} C_VEL
LIN {X 0,Y 573.33,Z 321.885,A -85,B 0,C 180,E1 -2160.703,E2 -2160.703} C_VEL
LIN {X 0,Y 573.241,Z 321.893,A -85,B 0,C 180,E1 -2163.515,E2 -2163.515} C_VEL
LIN {X 0,Y 573.283,Z 321.891,A -85,B 0,C 180,E1 -2165.629,E2 -2165.629} C_VEL
LIN {X 0,Y 573.277,Z 321.888,A -85,B 0,C 180,E1 -2168.46,E2 -2168.46} C_VEL
LIN {X 0,Y 573.289,Z 321.888,A -85,B 0,C 180,E1 -2171.312,E2 -2171.312} C_VEL
LIN {X 0,Y 573.272,Z 321.889,A -85,B 0,C 180,E1 -2174.426,E2 -2174.426} C_VEL
LIN {X 0,Y 573.252,Z 321.892,A -85,B 0,C 180,E1 -2177.112,E2 -2177.112} C_VEL
LIN {X 0,Y 573.246,Z 321.896,A -85,B 0,C 180,E1 -2180.077,E2 -2180.077} C_VEL
LIN {X 0,Y 573.225,Z 321.895,A -85,B 0,C 180,E1 -2183.1,E2 -2183.1} C_VEL
LIN {X 0,Y 573.246,Z 321.893,A -85,B 0,C 180,E1 -2185.411,E2 -2185.411} C_VEL
LIN {X 0,Y 573.257,Z 321.891,A -85,B 0,C 180,E1 -2188.033,E2 -2188.033} C_VEL
LIN {X 0,Y 573.227,Z 321.897,A -85,B 0,C 180,E1 -2190.884,E2 -2190.884} C_VEL
LIN {X 0,Y 573.281,Z 321.89,A -85,B 0,C 180,E1 -2193.529,E2 -2193.529} C_VEL
LIN {X 0,Y 573.255,Z 321.893,A -85,B 0,C 180,E1 -2196.049,E2 -2196.049} C_VEL
LIN {X 0,Y 573.243,Z 321.893,A -85,B 0,C 180,E1 -2198.702,E2 -2198.702} C_VEL
LIN {X 0,Y 573.246,Z 321.893,A -85,B 0,C 180,E1 -2201.597,E2 -2201.597} C_VEL
LIN {X 0,Y 573.233,Z 321.897,A -85,B 0,C 180,E1 -2204.334,E2 -2204.334} C_VEL
LIN {X 0,Y 573.237,Z 321.893,A -85,B 0,C 180,E1 -2207.359,E2 -2207.359} C_VEL
LIN {X 0,Y 573.242,Z 321.896,A -85,B 0,C 180,E1 -2210.394,E2 -2210.394} C_VEL
LIN {X 0,Y 573.252,Z 321.893,A -85,B 0,C 180,E1 -2213.079,E2 -2213.079} C_VEL
LIN {X 0,Y 573.301,Z 321.887,A -85,B 0,C 180,E1 -2216.1,E2 -2216.1} C_VEL
LIN {X 0,Y 573.322,Z 322.082,A -85,B 0,C 180,E1 -2216.523,E2 -2216.523} C_VEL
LIN {X 0,Y 573.646,Z 325.573,A -85,B 0,C 180,E1 -2217.71,E2 -2217.71} C_VEL
LIN {X 0,Y 573.499,Z 333.997,A -85,B 0,C 180,E1 -2220.468,E2 -2220.468} C_VEL
LIN {X 0,Y 573.383,Z 343.774,A -85,B 0,C 180,E1 -2223.479,E2 -2223.479} C_VEL
LIN {X 0,Y 573.339,Z 352.686,A -85,B 0,C 180,E1 -2226.141,E2 -2226.141} C_VEL
LIN {X 0,Y 573.255,Z 361.403,A -85,B 0,C 180,E1 -2228.709,E2 -2228.709} C_VEL
LIN {X 0,Y 573.179,Z 370.65,A -85,B 0,C 180,E1 -2231.411,E2 -2231.411} C_VEL
LIN {X 0,Y 573.153,Z 379.591,A -85,B 0,C 180,E1 -2233.986,E2 -2233.986} C_VEL
LIN {X 0,Y 573.095,Z 389.81,A -85,B 0,C 180,E1 -2236.888,E2 -2236.888} C_VEL
LIN {X 0,Y 573.051,Z 398.751,A -85,B 0,C 180,E1 -2239.4,E2 -2239.4} C_VEL
LIN {X 0,Y 573.034,Z 401.306,A -85,B 0,C 180,E1 -2240.114,E2 -2240.114} C_VEL
LIN {X 0,Y 573.514,Z 408.451,A -85,B 0,C 180,E1 -2240.301,E2 -2240.301} C_VEL
LIN {X 0,Y 573.46,Z 416.918,A -85,B 0,C 180,E1 -2240.567,E2 -2240.567} C_VEL
LIN {X 0,Y 573.401,Z 425.42,A -85,B 0,C 180,E1 -2240.921,E2 -2240.921} C_VEL
LIN {X 0,Y 573.335,Z 433.748,A -85,B 0,C 180,E1 -2241.365,E2 -2241.365} C_VEL
LIN {X 0,Y 573.249,Z 441.782,A -85,B 0,C 180,E1 -2241.896,E2 -2241.896} C_VEL
LIN {X 0,Y 573.193,Z 450.442,A -85,B 0,C 180,E1 -2242.604,E2 -2242.604} C_VEL
LIN {X 0,Y 573.151,Z 457.589,A -85,B 0,C 180,E1 -2243.327,E2 -2243.327} C_VEL
LIN {X 0,Y 573.112,Z 464.44,A -85,B 0,C 180,E1 -2244.194,E2 -2244.194} C_VEL
LIN {X 0,Y 572.995,Z 469.993,A -85,B 0,C 180,E1 -2245.076,E2 -2245.076} C_VEL
LIN {X 0,Y 573.036,Z 475.152,A -85,B 0,C 180,E1 -2246.133,E2 -2246.133} C_VEL
LIN {X 0,Y 572.99,Z 477.792,A -85,B 0,C 180,E1 -2246.837,E2 -2246.837} C_VEL
LIN {X 0,Y 572.94,Z 480.683,A -85,B 0,C 180,E1 -2247.892,E2 -2247.892} C_VEL
LIN {X 0,Y 572.944,Z 481.937,A -85,B 0,C 180,E1 -2248.595,E2 -2248.595} C_VEL
LIN {X 0,Y 572.937,Z 482.711,A -85,B 0,C 180,E1 -2249.298,E2 -2249.298} C_VEL
LIN {X 0,Y 572.935,Z 483,A -85,B 0,C 180,E1 -2250.001,E2 -2250.001} C_VEL
LIN {X 0,Y 572.937,Z 482.71,A -85,B 0,C 180,E1 -2250.704,E2 -2250.704} C_VEL
LIN {X 0,Y 572.944,Z 481.934,A -85,B 0,C 180,E1 -2251.407,E2 -2251.407} C_VEL
LIN {X 0,Y 572.94,Z 480.679,A -85,B 0,C 180,E1 -2252.11,E2 -2252.11} C_VEL
LIN {X 0,Y 572.99,Z 477.785,A -85,B 0,C 180,E1 -2253.165,E2 -2253.165} C_VEL
LIN {X 0,Y 573.024,Z 475.144,A -85,B 0,C 180,E1 -2253.869,E2 -2253.869} C_VEL
LIN {X 0,Y 572.995,Z 469.981,A -85,B 0,C 180,E1 -2254.926,E2 -2254.926} C_VEL
LIN {X 0,Y 573.138,Z 463.18,A -85,B 0,C 180,E1 -2255.984,E2 -2255.984} C_VEL
LIN {X 0,Y 573.165,Z 455.799,A -85,B 0,C 180,E1 -2256.86,E2 -2256.86} C_VEL
LIN {X 0,Y 573.216,Z 448.397,A -85,B 0,C 180,E1 -2257.575,E2 -2257.575} C_VEL
LIN {X 0,Y 573.274,Z 440.534,A -85,B 0,C 180,E1 -2258.194,E2 -2258.194} C_VEL
LIN {X 0,Y 573.382,Z 430.717,A -85,B 0,C 180,E1 -2258.814,E2 -2258.814} C_VEL
LIN {X 0,Y 573.433,Z 419.279,A -85,B 0,C 180,E1 -2259.347,E2 -2259.347} C_VEL
LIN {X 0,Y 573.521,Z 409.215,A -85,B 0,C 180,E1 -2259.679,E2 -2259.679} C_VEL
LIN {X 0,Y 573.228,Z 402.988,A -85,B 0,C 180,E1 -2259.84,E2 -2259.84} C_VEL
LIN {X 0,Y 573.035,Z 401.299,A -85,B 0,C 180,E1 -2259.888,E2 -2259.888} C_VEL
LIN {X 0,Y 573.08,Z 392.358,A -85,B 0,C 180,E1 -2262.394,E2 -2262.394} C_VEL
LIN {X 0,Y 573.146,Z 382.139,A -85,B 0,C 180,E1 -2265.287,E2 -2265.287} C_VEL
LIN {X 0,Y 573.206,Z 371.921,A -85,B 0,C 180,E1 -2268.22,E2 -2268.22} C_VEL
LIN {X 0,Y 573.258,Z 362.979,A -85,B 0,C 180,E1 -2270.827,E2 -2270.827} C_VEL
LIN {X 0,Y 573.318,Z 353.956,A -85,B 0,C 180,E1 -2273.479,E2 -2273.479} C_VEL
LIN {X 0,Y 573.373,Z 344.819,A -85,B 0,C 180,E1 -2276.185,E2 -2276.185} C_VEL
LIN {X 0,Y 573.444,Z 335.774,A -85,B 0,C 180,E1 -2278.954,E2 -2278.954} C_VEL
LIN {X 0,Y 573.623,Z 328.29,A -85,B 0,C 180,E1 -2281.38,E2 -2281.38} C_VEL
LIN {X 0,Y 573.504,Z 323.3,A -85,B 0,C 180,E1 -2283.048,E2 -2283.048} C_VEL
LIN {X 0,Y 573.284,Z 321.891,A -85,B 0,C 180,E1 -2283.577,E2 -2283.577} C_VEL
LIN {X 0,Y 573.257,Z 321.894,A -85,B 0,C 180,E1 -2286.923,E2 -2286.923} C_VEL
LIN {X 0,Y 573.24,Z 321.896,A -85,B 0,C 180,E1 -2289.608,E2 -2289.608} C_VEL
LIN {X 0,Y 573.248,Z 321.895,A -85,B 0,C 180,E1 -2292.642,E2 -2292.642} C_VEL
LIN {X 0,Y 573.227,Z 321.896,A -85,B 0,C 180,E1 -2295.665,E2 -2295.665} C_VEL
LIN {X 0,Y 573.234,Z 321.895,A -85,B 0,C 180,E1 -2298.543,E2 -2298.543} C_VEL
LIN {X 0,Y 573.242,Z 321.895,A -85,B 0,C 180,E1 -2301.298,E2 -2301.298} C_VEL
LIN {X 0,Y 573.218,Z 321.896,A -85,B 0,C 180,E1 -2304.019,E2 -2304.019} C_VEL
LIN {X 0,Y 573.242,Z 321.893,A -85,B 0,C 180,E1 -2306.516,E2 -2306.516} C_VEL
LIN {X 0,Y 573.228,Z 321.896,A -85,B 0,C 180,E1 -2309.119,E2 -2309.119} C_VEL
LIN {X 0,Y 573.241,Z 321.894,A -85,B 0,C 180,E1 -2311.435,E2 -2311.435} C_VEL
LIN {X 0,Y 573.266,Z 321.891,A -85,B 0,C 180,E1 -2313.81,E2 -2313.81} C_VEL
LIN {X 0,Y 573.232,Z 321.895,A -85,B 0,C 180,E1 -2316.134,E2 -2316.134} C_VEL
LIN {X 0,Y 573.254,Z 321.892,A -85,B 0,C 180,E1 -2319.173,E2 -2319.173} C_VEL
LIN {X 0,Y 573.221,Z 321.897,A -85,B 0,C 180,E1 -2321.411,E2 -2321.411} C_VEL
LIN {X 0,Y 573.253,Z 321.894,A -85,B 0,C 180,E1 -2323.621,E2 -2323.621} C_VEL
LIN {X 0,Y 573.235,Z 321.894,A -85,B 0,C 180,E1 -2326.529,E2 -2326.529} C_VEL
LIN {X 0,Y 573.269,Z 321.89,A -85,B 0,C 180,E1 -2328.745,E2 -2328.745} C_VEL
LIN {X 0,Y 573.258,Z 321.892,A -85,B 0,C 180,E1 -2331.54,E2 -2331.54} C_VEL
LIN {X 0,Y 573.292,Z 321.888,A -85,B 0,C 180,E1 -2334.371,E2 -2334.371} C_VEL
LIN {X 0,Y 573.308,Z 321.886,A -85,B 0,C 180,E1 -2337.892,E2 -2337.892} C_VEL
